REGION Network 6
   RUNG wire#powerrail
      #Module_Control(ReqUp := #Sequence_Control.ReqModulesUp, ReqDown := #Sequence_Control.ReqModulesDown, Sensor1Down := #Modules_DownPos1, Sensor1Up := #Modules_UpPos1, Sensor2Down := #Modules_DownPos2, Sensor2Up := #Modules_UpPos2, Interlock := true, Timeout :=, Valve => #Modules_Up, Error =>, "Step" =>, PosUp => #Module_Control.PosUp, PosDown => #Module_Control.PosDown)
   END_RUNG
   // the same network as SCL:
   #Module_Control(ReqUp := #Sequence_Control.ReqModulesUp,   // "CC_Vib_Modules"
                   ReqDown := #Sequence_Control.ReqModulesDown,
                   Sensor1Down := #Modules_DownPos1,
                   Sensor1Up := #Modules_UpPos1,
                   Sensor2Down := #Modules_DownPos2,
                   Sensor2Up := #Modules_UpPos2,
                   Interlock := true,
                   Valve => #Modules_Up,
                   PosUp => #Module_Control.PosUp,
                   PosDown => #Module_Control.PosDown);
END_REGION
END_FUNCTION_BLOCK

FUNCTION_BLOCK "CC_Sequence_Control"
{ S7_Optimized_Access := 'TRUE' }
VERSION : 0.1
   VAR_INPUT 
      Button_DriveRollers_Down : Bool;
      Button_DriveRollers_Up : Bool;
      Button_modules_Down : Bool;
      Button_modules_Up : Bool;
      Button_Pallete_Down : Bool;
      Button_Pallete_Up : Bool;
      Button_Wib : Bool;
      Seq_Forward : Bool;
      Seq_Backward : Bool;
      Drive_Rollers_DownPos : Bool;
      Drive_Rollers_UpPos : Bool;
      Pallete_DownPos : Bool;
      Pallete_UpPos : Bool;
      Modules_DownPos : Bool;
      Modules_UpPos : Bool;
      Centering_DownPos : Bool;
      Centering_UpPos : Bool;
   END_VAR

   VAR_OUTPUT 
      ReqPalleteUp : Bool;
      ReqPalleteDown : Bool;
      ReqDriveRollerUp : Bool;
      ReqDriveRollerDown : Bool;
      ReqModulesUp : Bool;
      ReqModulesDown : Bool;
      ReqVibrationEnable : Bool;
      Station_basePos : Bool;
   END_VAR

   VAR 
      Step { S7_SetPoint := 'True'} : Int;
      Button_Backward_TON {InstructionName := 'TON_TIME'; LibVersion := '1.0'} : TON_TIME;
   END_VAR

   VAR CONSTANT 
      sNOT_AUTOMATIC : Int;
      sBASE_POSITION : Int := 1;
      sMOVING_DRIVE_ROLLER : Int := 2;
      sMOVING_PALLETE : Int := 3;
      sMOVING_COMPACTION_MODULE : Int := 4;
      sCOMPACTING : Int := 5;
   END_VAR


BEGIN
	// Reset outputów
	#ReqPalleteUp := FALSE;
	#ReqPalleteDown := FALSE;
	#ReqDriveRollerUp := FALSE;
	#ReqDriveRollerDown := FALSE;
	#ReqVibrationEnable := FALSE;
	#ReqModulesUp := FALSE;
	#ReqModulesDown := FALSE;
	#Station_basePos := FALSE;
	
	IF #Button_DriveRollers_Down OR #Button_DriveRollers_Up OR #Button_Pallete_Down OR #Button_Pallete_Up OR #Button_modules_Down OR #Button_modules_Up OR #Button_Wib THEN
	    #Step := #sNOT_AUTOMATIC;
	ELSIF #Pallete_UpPos AND NOT #Seq_Forward AND #Drive_Rollers_UpPos AND #Modules_DownPos AND #Centering_DownPos THEN
	    #Step := #sBASE_POSITION;
	    #Station_basePos := true;
	END_IF;
	
	
	CASE #Step OF
	    #sBASE_POSITION:
	        IF #Seq_Forward THEN
	            #Step := #sMOVING_DRIVE_ROLLER;
	        END_IF;
	    #sMOVING_DRIVE_ROLLER:
	        #ReqPalleteUp := TRUE;
	        IF #Seq_Forward THEN
	            #ReqDriveRollerDown := TRUE;
	            IF #Drive_Rollers_DownPos THEN
	                #Step := #sMOVING_PALLETE;
	            END_IF;
	        ELSIF #Seq_Backward THEN
	            #ReqDriveRollerUp := TRUE;
	            IF #Drive_Rollers_UpPos THEN
	                #Step := #sBASE_POSITION;
	            END_IF;
	        END_IF;
	        
	    #sMOVING_PALLETE:
	        IF #Seq_Forward THEN
	            #ReqPalleteDown := TRUE;
	            IF #Pallete_DownPos THEN
	                #Step := #sMOVING_COMPACTION_MODULE;
	            END_IF;
	        ELSIF #Seq_Backward THEN
	            #ReqPalleteUp := TRUE;
	            IF #Pallete_UpPos THEN
	                #Step := #sMOVING_DRIVE_ROLLER;
	            END_IF;
	        END_IF;
	        
	    #sMOVING_COMPACTION_MODULE:
	        IF #Seq_Forward THEN
	            #ReqModulesUp := TRUE;
	         //   IF #Modules_UpPos THEN
	                #Step := #sCOMPACTING;
	         //   END_IF;
	        ELSIF #Seq_Backward THEN
	            #ReqModulesDown := TRUE;
	            IF #Modules_DownPos THEN
	                #Step := #sMOVING_PALLETE;
	            END_IF;
	        END_IF;
	        
	    #sCOMPACTING:
	        // Warunek zakończenia kompaktowania (np. czas lub czujnik)
	        IF #Seq_Forward THEN
	            #ReqVibrationEnable := TRUE;
	            #Step := #sCOMPACTING;
	        ELSIF #Seq_Backward THEN
	            #Step := #sMOVING_COMPACTION_MODULE;
	        END_IF;
	        
	    #sNOT_AUTOMATIC:
	        #ReqDriveRollerDown := #Button_DriveRollers_Down;
	        #ReqDriveRollerUp := #Button_DriveRollers_Up;
	        #ReqModulesDown := #Button_modules_Down;
	        #ReqModulesUp := #Button_modules_Up;
	        #ReqPalleteDown := #Button_Pallete_Down;
	        #ReqPalleteUp := #Button_Pallete_Up;
	        #ReqVibrationEnable := #Button_Wib;
	        
	END_CASE;
END_FUNCTION_BLOCK

FUNCTION_BLOCK "CC_Hydraulic_Rollers"   // FB101, LAD
{ S7_Optimized_Access := 'TRUE' }
// stored: AutoNumber false, MemoryReserve 100, SetENOAutomatically false
   VAR_INPUT
      ReqUp : Bool;
      ReqDown : Bool;
      Sensor1Down : Bool;
      Sensor1Up : Bool;
      Sensor2Down : Bool;
      Sensor2Up : Bool;
      InterlockMove : Bool;
      HydUnitReady : Bool;
   END_VAR
   VAR_OUTPUT
      HydraulicUnit : Bool;
      ValveUp : Bool;
      ValveDown : Bool;
      error : Byte;   // %X0 – nieprawidłowa pozycja dolna %X1 nieprawidłowa pozycja górna %X2 – przekroczony czas ruchu
      "Step" : Int;
      PosUp : Bool;
      PosDown : Bool;
   END_VAR
   VAR
      IEC_Extention { S7_SetPoint := 'True'} : TON_TIME;
      IEC_RETRACTION { S7_SetPoint := 'True'} : TON_TIME;
      tMotionTimeout { S7_SetPoint := 'True'} : TON_TIME;
   END_VAR
   VAR CONSTANT
      STEP_RETRACT : Int := 1;
      STEP_MOVING : Int := 2;
      STEP_EXTEND : Int := 3;
   END_VAR
BEGIN

REGION Network 1: ValveUp
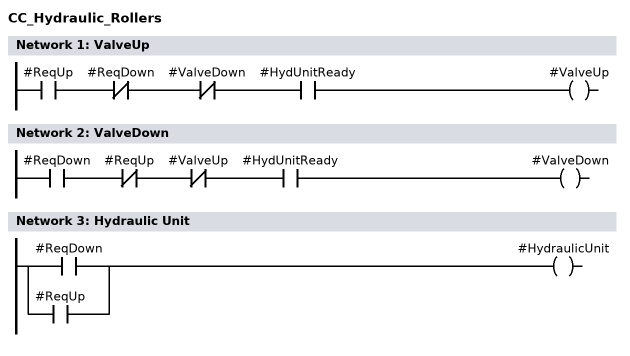
   RUNG wire#powerrail
      Contact( #ReqUp )
      I_Contact( #ReqDown )
      I_Contact( #ValveDown )
      Contact( #HydUnitReady )
      Coil( #ValveUp )
   END_RUNG
   // the same network as SCL:
   #ValveUp := #ReqUp AND NOT #ReqDown AND NOT #ValveDown AND #HydUnitReady;
END_REGION

REGION Network 2: ValveDown
   RUNG wire#powerrail
      Contact( #ReqDown )
      I_Contact( #ReqUp )
      I_Contact( #ValveUp )
      Contact( #HydUnitReady )
      Coil( #ValveDown )
   END_RUNG
   // the same network as SCL:
   #ValveDown := #ReqDown AND NOT #ReqUp AND NOT #ValveUp AND #HydUnitReady;
END_REGION

REGION Network 3: Hydraulic Unit
   RUNG wire#powerrail
      Contact( #ReqDown )
      wire#w1
      Coil( #HydraulicUnit )
   END_RUNG
   RUNG wire#powerrail
      Contact( #ReqUp )
   END_RUNG wire#w1
   // the same network as SCL:
   #HydraulicUnit := #ReqDown OR #ReqUp;
END_REGION

REGION Network 4 (SCL)
   #PosDown := false;
   #PosUp := FALSE;
   #Step := 0;
   IF #Sensor1Down = 0 AND #Sensor1Up = 1 AND #Sensor2Down = 0 AND #Sensor2Up = 1 THEN
       #Step.%X3 := TRUE;
       #PosUp := True;
   ELSIF #Sensor1Down = 1 AND #Sensor1Up =0 AND #Sensor2Down =1 AND #Sensor2Up =0 THEN
       #Step.%X1:= TRUE;
       #PosDown := True;
   ELSE
       #Step.%X2 := TRUE;
   END_IF;
END_REGION
END_FUNCTION_BLOCK

FUNCTION_BLOCK "CC_Pneumatic_Roller"   // FB104, LAD
{ S7_Optimized_Access := 'TRUE' }
// stored: AutoNumber false, MemoryReserve 100, SetENOAutomatically false
   VAR_INPUT
      ReqUp : Bool;
      ReqDown : Bool;
      Sensor1Down : Bool;
      Sensor1Up : Bool;
      Sensor2Down : Bool;
      Sensor2Up : Bool;
      Interlock : Bool;
      Timeout : Time := T#3s;
   END_VAR
   VAR_OUTPUT
      Valve : Bool;
      Error : Bool;
      "Step" : Int;
      PosUp : Bool;
      PosDown : Bool;
   END_VAR
   VAR
      IEC_Timout_retracting { S7_SetPoint := 'True'} : TOF_TIME;
      IEC_Timout_extracting { S7_SetPoint := 'True'} : TON_TIME;
   END_VAR
   VAR CONSTANT
      STEP_RETRACT : Int := 1;
      STEP_MOVING : Int := 2;
      STEP_EXTEND : Int := 3;
   END_VAR
BEGIN

REGION Network 1
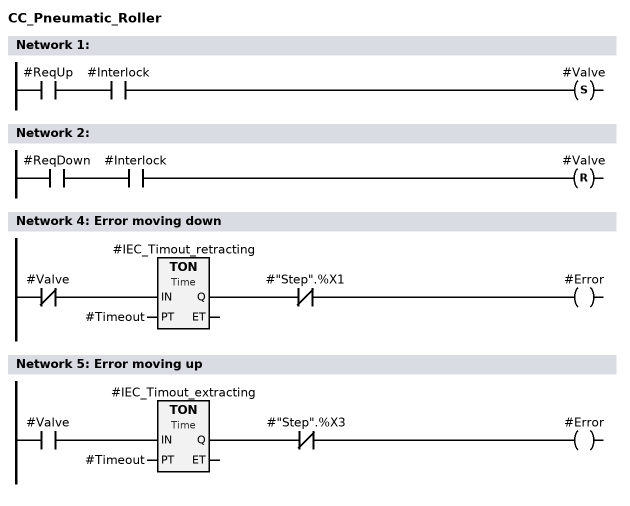
   RUNG wire#powerrail
      Contact( #ReqUp )
      Contact( #Interlock )
      S_Coil( #Valve )
   END_RUNG
   // the same network as SCL:
   IF #ReqUp AND #Interlock THEN #Valve := TRUE; END_IF;
END_REGION

REGION Network 2
   RUNG wire#powerrail
      Contact( #ReqDown )
      Contact( #Interlock )
      R_Coil( #Valve )
   END_RUNG
   // the same network as SCL:
   IF #ReqDown AND #Interlock THEN #Valve := FALSE; END_IF;
END_REGION

REGION Network 3 (SCL)
   #PosDown := FALSE;
   #PosUp := FALSE;
   #Step := 0;
   IF #Sensor1Down = 0 AND #Sensor1Up = 1 AND #Sensor2Down = 0 AND #Sensor2Up = 1 THEN
       #Step.%X3 :=1;
       #PosUp := True;
   ELSIF #Sensor1Down AND #Sensor1Up = 0 AND #Sensor2Down AND #Sensor2Up = 0 THEN
       #Step.%X1 := 1;
       #PosDown := True;
   ELSE
       #Step.%X2:= 1;
   END_IF;
END_REGION

REGION Network 4: Error moving down
   RUNG wire#powerrail
      I_Contact( #Valve )
      { S7_Templates := "time_type := Time" } #IEC_Timout_retracting.TON(pt := #Timeout, et =>)
      I_Contact( #"Step".%X1 )
      Coil( #Error )
   END_RUNG
   // the same network as SCL:
   #IEC_Timout_retracting(IN := NOT #Valve, PT := #Timeout);   // TON
   #Error := #IEC_Timout_retracting.Q AND NOT #"Step".%X1;
END_REGION

REGION Network 5: Error moving up
   RUNG wire#powerrail
      Contact( #Valve )
      { S7_Templates := "time_type := Time" } #IEC_Timout_extracting.TON(pt := #Timeout, et =>)
      I_Contact( #"Step".%X3 )
      Coil( #Error )
   END_RUNG
   // the same network as SCL:
   #IEC_Timout_extracting(IN := #Valve, PT := #Timeout);   // TON
   #Error := #IEC_Timout_extracting.Q AND NOT #"Step".%X3;
END_REGION
END_FUNCTION_BLOCK

FUNCTION_BLOCK "CC_Vib_Modules"   // FB102, LAD
{ S7_Optimized_Access := 'TRUE' }
// stored: AutoNumber false, MemoryReserve 100, SetENOAutomatically false
   VAR_INPUT
      ReqUp : Bool;
      ReqDown : Bool;
      Sensor1Down : Bool;
      Sensor1Up : Bool;
      Sensor2Down : Bool;
      Sensor2Up : Bool;
      Interlock : Bool := false;
      Timeout : Time := T#3s;
   END_VAR
   VAR_OUTPUT
      Valve : Bool;
      Error : Bool;
      "Step" : Int;
      PosUp : Bool;
      PosDown : Bool;
   END_VAR
   VAR
      IEC_Timout_retracting { S7_SetPoint := 'True'} : TOF_TIME;
      IEC_Timout_extracting { S7_SetPoint := 'True'} : TON_TIME;
   END_VAR
   VAR CONSTANT
      STEP_RETRACT : Int := 1;
      STEP_MOVING : Int := 2;
      STEP_EXTEND : Int := 3;
   END_VAR
BEGIN

REGION Network 1
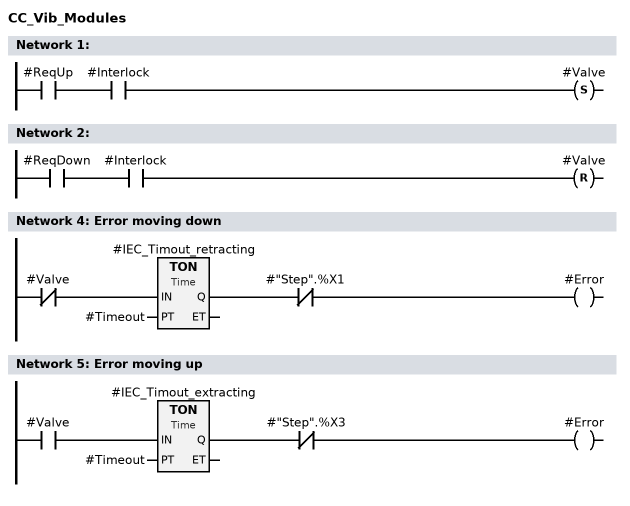
   RUNG wire#powerrail
      Contact( #ReqUp )
      Contact( #Interlock )
      S_Coil( #Valve )
   END_RUNG
   // the same network as SCL:
   IF #ReqUp AND #Interlock THEN #Valve := TRUE; END_IF;
END_REGION

REGION Network 2
   RUNG wire#powerrail
      Contact( #ReqDown )
      Contact( #Interlock )
      R_Coil( #Valve )
   END_RUNG
   // the same network as SCL:
   IF #ReqDown AND #Interlock THEN #Valve := FALSE; END_IF;
END_REGION

REGION Network 3 (SCL)
   #PosDown := false;
   #PosUp := false;
   #Step := 0;
   IF #Sensor1Down = 0 AND #Sensor1Up = 1 AND #Sensor2Down = 0 AND #Sensor2Up = 1 THEN
       #Step.%X3 := TRUE;
       #PosUp := True;
   ELSIF #Sensor1Down AND #Sensor1Up AND #Sensor2Down AND #Sensor2Up THEN
       #Step.%X1 := TRUE;
       #PosDown := True;
   ELSE
       #Step.%X2 := TRUE;
   END_IF;
END_REGION

REGION Network 4: Error moving down
   RUNG wire#powerrail
      I_Contact( #Valve )
      { S7_Templates := "time_type := Time" } #IEC_Timout_retracting.TON(pt := #Timeout, et =>)
      I_Contact( #"Step".%X1 )
      Coil( #Error )
   END_RUNG
   // the same network as SCL:
   #IEC_Timout_retracting(IN := NOT #Valve, PT := #Timeout);   // TON
   #Error := #IEC_Timout_retracting.Q AND NOT #"Step".%X1;
END_REGION

REGION Network 5: Error moving up
   RUNG wire#powerrail
      Contact( #Valve )
      { S7_Templates := "time_type := Time" } #IEC_Timout_extracting.TON(pt := #Timeout, et =>)
      I_Contact( #"Step".%X3 )
      Coil( #Error )
   END_RUNG
   // the same network as SCL:
   #IEC_Timout_extracting(IN := #Valve, PT := #Timeout);   // TON
   #Error := #IEC_Timout_extracting.Q AND NOT #"Step".%X3;
END_REGION
END_FUNCTION_BLOCK

FUNCTION_BLOCK "CC_Vibrator_Control"   // FB103, LAD
{ S7_Optimized_Access := 'TRUE' }
// stored: AutoNumber false, MemoryReserve 100, SetENOAutomatically false
   VAR_INPUT
      StartVibrating : Bool;
      Reset : Bool;
      Axis : TO_SpeedAxis;
      tmpVelocity : LReal := 2840.0;
   END_VAR
   VAR
      MC_Power_data { S7_SetPoint := 'True'} : MC_POWER;
      MC_Reset_data { S7_SetPoint := 'True'} : MC_RESET;
      MC_MoveJog_data { S7_SetPoint := 'True'} : MC_MOVEJOG;
      MC_HALT_data { S7_SetPoint := 'True'} : MC_HALT;
   END_VAR
BEGIN

REGION Network 1: Hydraulic Unit Motion Control
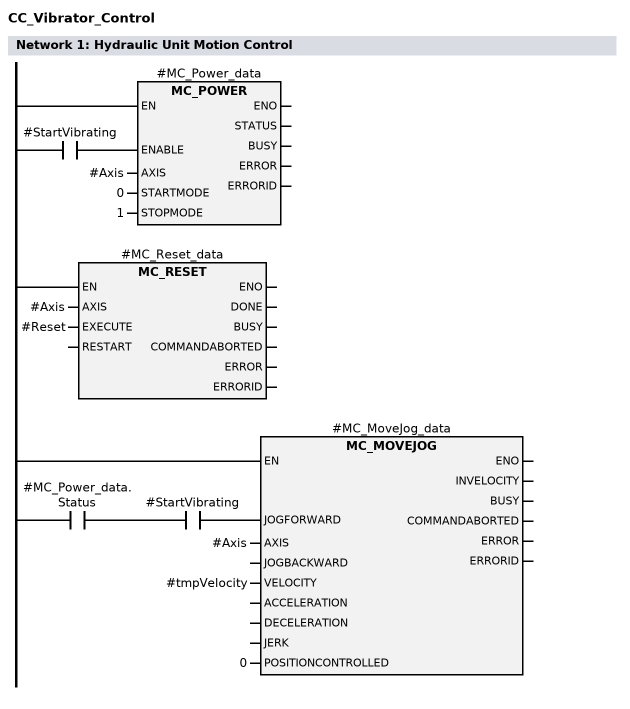
   RUNG wire#powerrail
      #MC_Power_data.MC_POWER(Enable := wire#w1, Axis := #Axis, StartMode := 0, StopMode := 1, Status =>, Busy =>, Error =>, ErrorId =>)
   END_RUNG
   RUNG wire#powerrail
      Contact( #StartVibrating )
   END_RUNG wire#w1
   RUNG wire#powerrail
      #MC_Reset_data.MC_RESET(Axis := #Axis, Execute := #Reset, Restart :=, Done =>, Busy =>, CommandAborted =>, Error =>, ErrorId =>)
   END_RUNG
   RUNG wire#powerrail
      #MC_MoveJog_data.MC_MOVEJOG(JogForward := wire#w2, Axis := #Axis, JogBackward :=, Velocity := #tmpVelocity, Acceleration :=, Deceleration :=, Jerk :=, PositionControlled := 0, InVelocity =>, Busy =>, CommandAborted =>, Error =>, ErrorId =>)
   END_RUNG
   RUNG wire#powerrail
      Contact( #MC_Power_data.Status )
      Contact( #StartVibrating )
   END_RUNG wire#w2
   // the same network as SCL:
   #MC_Power_data(Enable := #StartVibrating, Axis := #Axis, StartMode := 0, StopMode := 1);   // MC_POWER
   #MC_Reset_data(Axis := #Axis, Execute := #Reset);   // MC_RESET
   #MC_MoveJog_data(JogForward := #MC_Power_data.Status AND #StartVibrating,   // MC_MOVEJOG
                    Axis := #Axis,
                    Velocity := #tmpVelocity,
                    PositionControlled := 0);
END_REGION
END_FUNCTION_BLOCK

FUNCTION_BLOCK "Oil"   // FB8, LAD
{ S7_Optimized_Access := 'TRUE' }
// stored: MemoryReserve 100, SetENOAutomatically false
   VAR_INPUT
      Safety_OK : Bool;
      Pump_status : Bool;
      Pump_error : Bool;
      Pallette_Moving : Bool;
   END_VAR
   VAR_OUTPUT
      Pump : Bool;
      Main_Valve : Bool;
      Preparation_Valve : Bool;
      Nozzle_Valve : Bool;
      Pump_Volume_Output : Int;
   END_VAR
   VAR
      Pump_Reset { S7_SetPoint := 'True'} : TON_TIME;
      Pump_Volume { S7_SetPoint := 'True'} : Real;
      Oil_Station_Enable : Bool;
   END_VAR
   VAR_TEMP
      tmp : Int;
   END_VAR
BEGIN

REGION Network 1
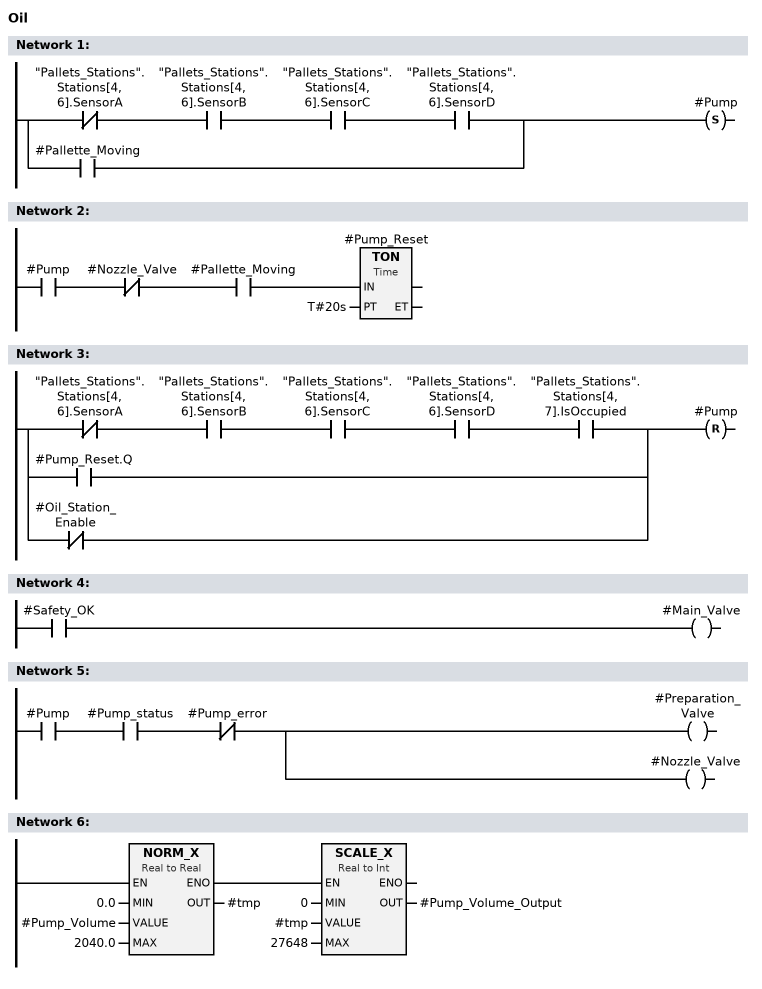
   RUNG wire#powerrail
      I_Contact( "Pallets_Stations".Stations[4, 6].SensorA )
      Contact( "Pallets_Stations".Stations[4, 6].SensorB )
      Contact( "Pallets_Stations".Stations[4, 6].SensorC )
      Contact( "Pallets_Stations".Stations[4, 6].SensorD )
      wire#w1
      S_Coil( #Pump )
   END_RUNG
   RUNG wire#powerrail
      Contact( #Pallette_Moving )
   END_RUNG wire#w1
   // the same network as SCL:
   IF (NOT "Pallets_Stations".Stations[4, 6].SensorA AND "Pallets_Stations".Stations[4, 6].SensorB AND "Pallets_Stations".Stations[4, 6].SensorC AND "Pallets_Stations".Stations[4, 6].SensorD) OR #Pallette_Moving THEN
       #Pump := TRUE;
   END_IF;
END_REGION

REGION Network 2
   RUNG wire#powerrail
      Contact( #Pump )
      I_Contact( #Nozzle_Valve )
      Contact( #Pallette_Moving )
      { S7_Templates := "time_type := Time" } #Pump_Reset.TON(pt := T#20s, et =>)
   END_RUNG
   // the same network as SCL:
   #Pump_Reset(IN := #Pump AND NOT #Nozzle_Valve AND #Pallette_Moving, PT := T#20s);   // TON
END_REGION

REGION Network 3
   RUNG wire#powerrail
      I_Contact( "Pallets_Stations".Stations[4, 6].SensorA )
      Contact( "Pallets_Stations".Stations[4, 6].SensorB )
      Contact( "Pallets_Stations".Stations[4, 6].SensorC )
      Contact( "Pallets_Stations".Stations[4, 6].SensorD )
      Contact( "Pallets_Stations".Stations[4, 7].IsOccupied )
      wire#w1
      R_Coil( #Pump )
   END_RUNG
   RUNG wire#powerrail
      Contact( #Pump_Reset.Q )
   END_RUNG wire#w1
   RUNG wire#powerrail
      I_Contact( #Oil_Station_Enable )
   END_RUNG wire#w1
   // the same network as SCL:
   IF (NOT "Pallets_Stations".Stations[4, 6].SensorA AND "Pallets_Stations".Stations[4, 6].SensorB AND "Pallets_Stations".Stations[4, 6].SensorC AND "Pallets_Stations".Stations[4, 6].SensorD AND "Pallets_Stations".Stations[4, 7].IsOccupied) OR #Pump_Reset.Q OR NOT #Oil_Station_Enable THEN
       #Pump := FALSE;
   END_IF;
END_REGION

REGION Network 4
   RUNG wire#powerrail
      Contact( #Safety_OK )
      Coil( #Main_Valve )
   END_RUNG
   // the same network as SCL:
   #Main_Valve := #Safety_OK;
END_REGION

REGION Network 5
   RUNG wire#powerrail
      Contact( #Pump )
      Contact( #Pump_status )
      I_Contact( #Pump_error )
      wire#w1
      Coil( #Preparation_Valve )
   END_RUNG
   RUNG wire#w1
      Coil( #Nozzle_Valve )
   END_RUNG
   // the same network as SCL:
   #Preparation_Valve := #Pump AND #Pump_status AND NOT #Pump_error;
   #Nozzle_Valve := #Preparation_Valve;
END_REGION

REGION Network 6
   RUNG wire#powerrail
      { S7_Templates := "[SrcType := Real, DestType := Real]" } Normalize(min := 0.0, value := #Pump_Volume, max := 2040.0, out => #tmp)
      { S7_Templates := "[SrcType := Real, DestType := Int]" } Scale(min := 0, value := #tmp, max := 27648, out => #Pump_Volume_Output)
   END_RUNG
   // the same network as SCL:
   #tmp := NORM_X(MIN := 0.0, VALUE := #Pump_Volume, MAX := 2040.0);
   #Pump_Volume_Output := SCALE_X(MIN := 0, VALUE := #tmp, MAX := 27648);
END_REGION
END_FUNCTION_BLOCK

FUNCTION_BLOCK "HMI_Test"
{ S7_Optimized_Access := 'TRUE' }
VERSION : 0.1
   VAR 
      Old_Value : USInt;
      HMI_Connection_Alarm : Bool;
      Timer_2s {InstructionName := 'TON_TIME'; LibVersion := '1.0'; S7_SetPoint := 'False'} : TON_TIME;
   END_VAR


BEGIN
	IF #Timer_2s.Q THEN
	    #HMI_Connection_Alarm := ("HMI_DB".Heart_Bit = #Old_Value);
	    #Old_Value := "HMI_DB".Heart_Bit;
	END_IF;
	
	#Timer_2s(IN := NOT #Timer_2s.Q,
	          PT := T#2s);
	
END_FUNCTION_BLOCK

ORGANIZATION_BLOCK "CyclicInterrupt"   // OB30, LAD, CyclicInterrupt
{ S7_Optimized_Access := 'TRUE' }
// stored: SetENOAutomatically false
   VAR_INPUT
      Initial_Call : Bool;   // Initial call of this OB
      Event_Count : Int;   // Events discarded
   END_VAR
BEGIN

REGION Network 1
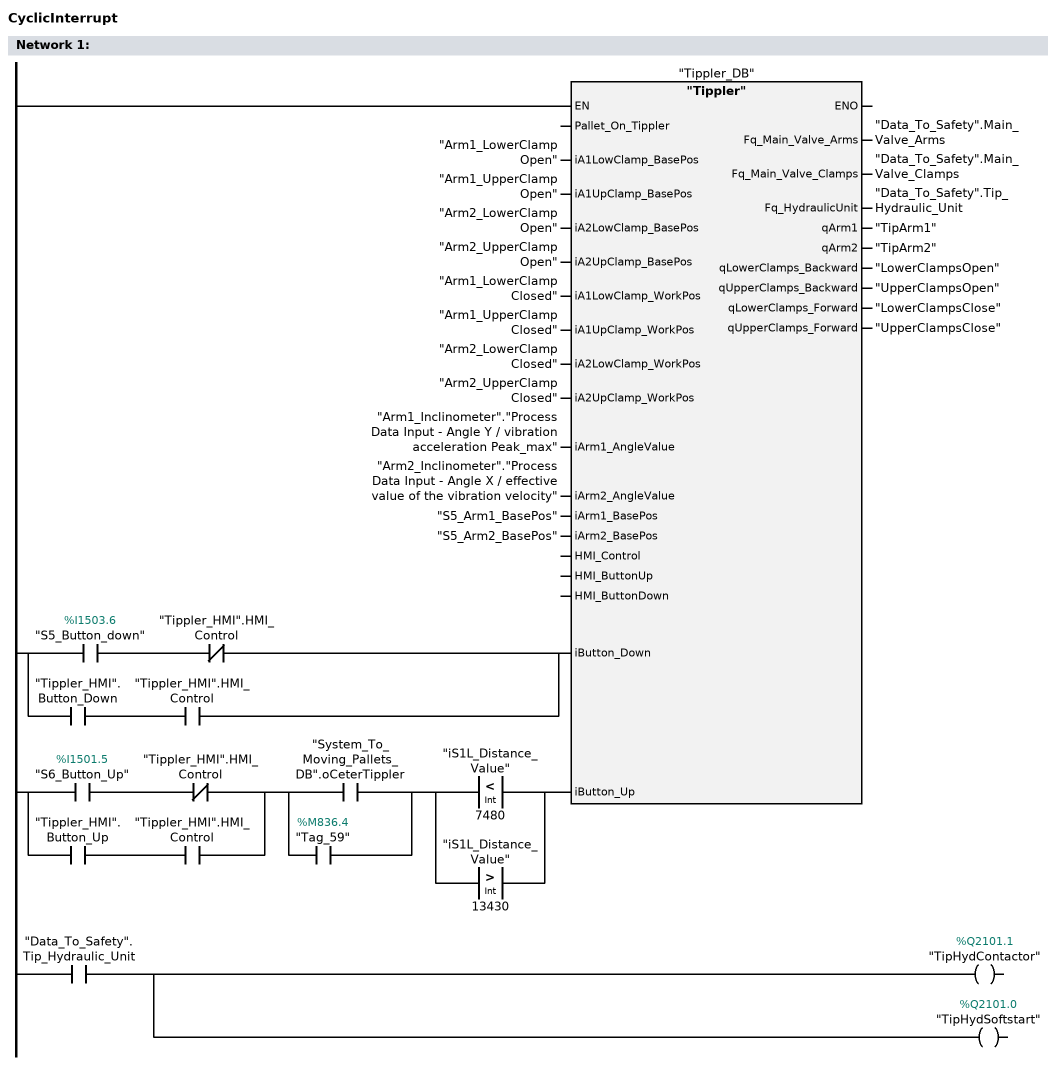
   RUNG wire#powerrail
      "Tippler_DB"(iButton_Down := wire#w1, iButton_Up := wire#w4, Pallet_On_Tippler :=, iA1LowClamp_BasePos := "Arm1_LowerClampOpen", iA1UpClamp_BasePos := "Arm1_UpperClampOpen", iA2LowClamp_BasePos := "Arm2_LowerClampOpen", iA2UpClamp_BasePos := "Arm2_UpperClampOpen", iA1LowClamp_WorkPos := "Arm1_LowerClampClosed", iA1UpClamp_WorkPos := "Arm1_UpperClampClosed", iA2LowClamp_WorkPos := "Arm2_LowerClampClosed", iA2UpClamp_WorkPos := "Arm2_UpperClampClosed", iArm1_AngleValue := "Arm1_Inclinometer"."Process Data Input - Angle Y / vibration acceleration Peak_max", iArm2_AngleValue := "Arm2_Inclinometer"."Process Data Input - Angle X / effective value of the vibration velocity", iArm1_BasePos := "S5_Arm1_BasePos", iArm2_BasePos := "S5_Arm2_BasePos", HMI_Control :=, HMI_ButtonUp :=, HMI_ButtonDown :=, Fq_Main_Valve_Arms => "Data_To_Safety".Main_Valve_Arms, Fq_Main_Valve_Clamps => "Data_To_Safety".Main_Valve_Clamps, Fq_HydraulicUnit => "Data_To_Safety".Tip_Hydraulic_Unit, qArm1 => "TipArm1", qArm2 => "TipArm2", qLowerClamps_Backward => "LowerClampsOpen", qUpperClamps_Backward => "UpperClampsOpen", qLowerClamps_Forward => "LowerClampsClose", qUpperClamps_Forward => "UpperClampsClose")
   END_RUNG
   RUNG wire#powerrail
      Contact( "S5_Button_down" )
      I_Contact( "Tippler_HMI".HMI_Control )
   END_RUNG wire#w1
   RUNG wire#powerrail
      Contact( "Tippler_HMI".Button_Down )
      Contact( "Tippler_HMI".HMI_Control )
   END_RUNG wire#w1
   RUNG wire#powerrail
      Contact( "S6_Button_Up" )
      I_Contact( "Tippler_HMI".HMI_Control )
      wire#w2
      Contact( "System_To_Moving_Pallets_DB".oCeterTippler )
      wire#w3
      { S7_Templates := "SrcType := Int" } LT_Contact(in1 := "iS1L_Distance_Value", in2 := 7480)
   END_RUNG wire#w4
   RUNG wire#powerrail
      Contact( "Tippler_HMI".Button_Up )
      Contact( "Tippler_HMI".HMI_Control )
   END_RUNG wire#w2
   RUNG wire#w2
      Contact( "Tag_59" )
   END_RUNG wire#w3
   RUNG wire#w3
      { S7_Templates := "SrcType := Int" } GT_Contact(in1 := "iS1L_Distance_Value", in2 := 13430)
   END_RUNG wire#w4
   RUNG wire#powerrail
      Contact( "Data_To_Safety".Tip_Hydraulic_Unit )
      wire#w5
      Coil( "TipHydContactor" )
   END_RUNG
   RUNG wire#w5
      Coil( "TipHydSoftstart" )
   END_RUNG
   // the same network as SCL:
   "Tippler_DB"(iA1LowClamp_BasePos := "Arm1_LowerClampOpen",   // "Tippler"
                iA1UpClamp_BasePos := "Arm1_UpperClampOpen",
                iA2LowClamp_BasePos := "Arm2_LowerClampOpen",
                iA2UpClamp_BasePos := "Arm2_UpperClampOpen",
                iA1LowClamp_WorkPos := "Arm1_LowerClampClosed",
                iA1UpClamp_WorkPos := "Arm1_UpperClampClosed",
                iA2LowClamp_WorkPos := "Arm2_LowerClampClosed",
                iA2UpClamp_WorkPos := "Arm2_UpperClampClosed",
                iArm1_AngleValue := "Arm1_Inclinometer"."Process Data Input - Angle Y / vibration acceleration Peak_max",
                iArm2_AngleValue := "Arm2_Inclinometer"."Process Data Input - Angle X / effective value of the vibration velocity",
                iArm1_BasePos := "S5_Arm1_BasePos",
                iArm2_BasePos := "S5_Arm2_BasePos",
                iButton_Down := ("S5_Button_down" AND NOT "Tippler_HMI".HMI_Control) OR ("Tippler_HMI".Button_Down AND "Tippler_HMI".HMI_Control),
                iButton_Up := (("S6_Button_Up" AND NOT "Tippler_HMI".HMI_Control) OR ("Tippler_HMI".Button_Up AND "Tippler_HMI".HMI_Control)) AND ("System_To_Moving_Pallets_DB".oCeterTippler OR "Tag_59") AND (("iS1L_Distance_Value" < 7480) OR ("iS1L_Distance_Value" > 13430)),
                Fq_Main_Valve_Arms => "Data_To_Safety".Main_Valve_Arms,
                Fq_Main_Valve_Clamps => "Data_To_Safety".Main_Valve_Clamps,
                Fq_HydraulicUnit => "Data_To_Safety".Tip_Hydraulic_Unit,
                qArm1 => "TipArm1",
                qArm2 => "TipArm2",
                qLowerClamps_Backward => "LowerClampsOpen",
                qUpperClamps_Backward => "UpperClampsOpen",
                qLowerClamps_Forward => "LowerClampsClose",
                qUpperClamps_Forward => "UpperClampsClose");
   "TipHydContactor" := "Data_To_Safety".Tip_Hydraulic_Unit;
   "TipHydSoftstart" := "Data_To_Safety".Tip_Hydraulic_Unit;
END_REGION
END_ORGANIZATION_BLOCK

FUNCTION_BLOCK "Tippler"   // FB400, LAD
{ S7_Optimized_Access := 'TRUE' }
// stored: AutoNumber false, MemoryReserve 100, SetENOAutomatically false
   VAR_INPUT
      Pallet_On_Tippler : Bool;
      iA1LowClamp_BasePos : Bool;
      iA1UpClamp_BasePos : Bool;
      iA2LowClamp_BasePos : Bool;
      iA2UpClamp_BasePos : Bool;
      iA1LowClamp_WorkPos : Bool;
      iA1UpClamp_WorkPos : Bool;
      iA2LowClamp_WorkPos : Bool;
      iA2UpClamp_WorkPos : Bool;
      iArm1_AngleValue : Int;
      iArm2_AngleValue : Int;
      iArm1_BasePos : Bool;
      iArm2_BasePos : Bool;
      HMI_Control : Bool;
      HMI_ButtonUp : Bool;
      HMI_ButtonDown : Bool;
      iButton_Down : Bool;
      iButton_Up : Bool;
   END_VAR
   VAR_OUTPUT
      Fq_Main_Valve_Arms : Bool;
      Fq_Main_Valve_Clamps : Bool;
      Fq_HydraulicUnit : Bool;
      qArm1 : Int;
      qArm2 : Int;
      qLowerClamps_Backward : Bool;
      qUpperClamps_Backward : Bool;
      qLowerClamps_Forward : Bool;
      qUpperClamps_Forward : Bool;
   END_VAR
   VAR
      Hydraulic_Ready { S7_SetPoint := 'True'} : TON_TIME;
      Hydraulic_Off { S7_SetPoint := 'True'} : TON_TIME;
      LowerClamps { S7_SetPoint := 'True'} : "Clamp";
      UpperClamps { S7_SetPoint := 'True'} : "Clamp";
      Arms { S7_SetPoint := 'True'} : "Arms";
      "Step" { S7_SetPoint := 'True'} : Int;
      ReqArmsDown : Bool;
      ReqArmsUp : Bool;
      Arms_workPos : Bool;
      Arms_basePos : Bool;
      Arms_clampsOperPos { S7_SetPoint := 'True'} : Bool;
      Tippler_maintenance { S7_SetPoint := 'True'} : "Tippler_maintenance";
      ButtonArmsDown { S7_SetPoint := 'True'} : Bool;
      ButtonArmsUp { S7_SetPoint := 'True'} : Bool;
      ReqLowerClampsClose : Bool;
      ReqUpperClampsClose : Bool;
      ReqLowerClampsOpen : Bool;
      ReqUpperClampsOpen : Bool;
      Timer_ClampsWorkPos { S7_SetPoint := 'True'} : TON_TIME;
      Timer_ClampsBasePos { S7_SetPoint := 'True'} : TON_TIME;
      Tippler_keep_down { S7_SetPoint := 'True'} : TP_TIME;
      N_Trig_Button_Down { S7_SetPoint := 'True'} : Bool;
   END_VAR
   VAR_TEMP
      Arm_Valves_Not_Actuated : Bool;
      Clamp_Valves_Not_Actuated : Bool;
   END_VAR
   VAR_TEMP   // added for the SCL form of the ladder/FBD networks
      _w1 : Bool;
   END_VAR
BEGIN

REGION Network 1: Zawory na ramionach niewysterowane
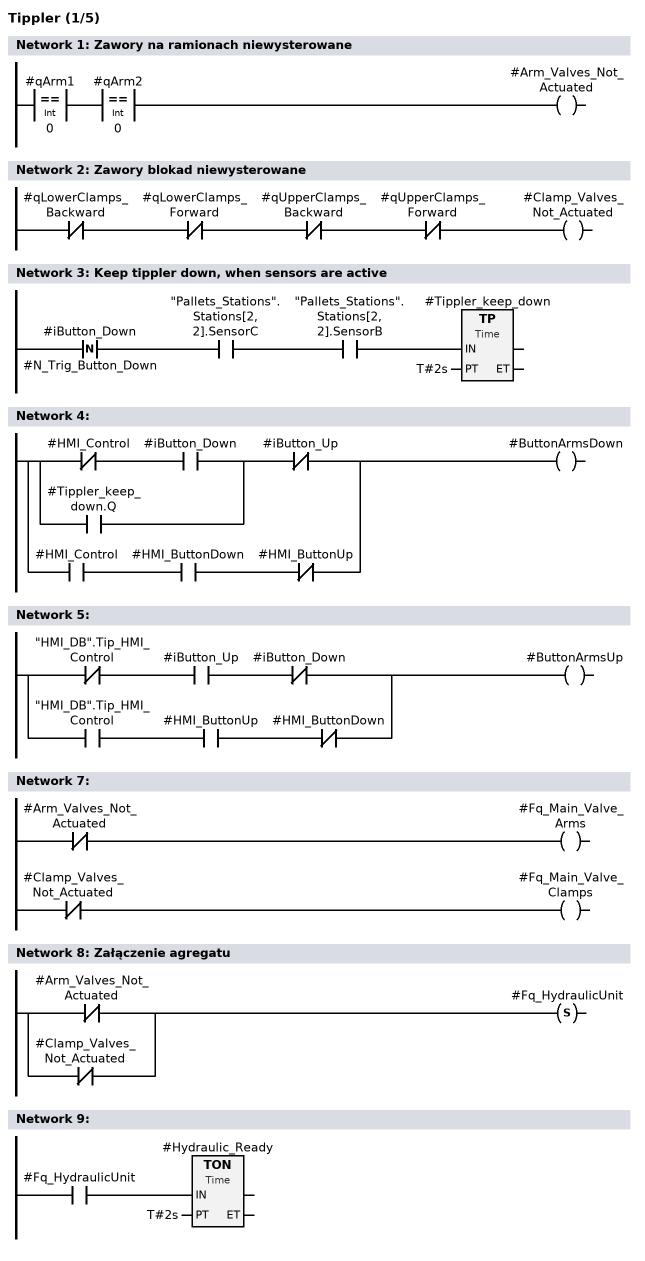
   RUNG wire#powerrail
      { S7_Templates := "SrcType := Int" } EQ_Contact(in1 := #qArm1, in2 := 0)
      { S7_Templates := "SrcType := Int" } EQ_Contact(in1 := #qArm2, in2 := 0)
      Coil( #Arm_Valves_Not_Actuated )
   END_RUNG
   // the same network as SCL:
   #Arm_Valves_Not_Actuated := (#qArm1 = 0) AND (#qArm2 = 0);
END_REGION

REGION Network 2: Zawory blokad niewysterowane
   RUNG wire#powerrail
      I_Contact( #qLowerClamps_Backward )
      I_Contact( #qLowerClamps_Forward )
      I_Contact( #qUpperClamps_Backward )
      I_Contact( #qUpperClamps_Forward )
      Coil( #Clamp_Valves_Not_Actuated )
   END_RUNG
   // the same network as SCL:
   #Clamp_Valves_Not_Actuated := NOT #qLowerClamps_Backward AND NOT #qLowerClamps_Forward AND NOT #qUpperClamps_Backward AND NOT #qUpperClamps_Forward;
END_REGION

REGION Network 3: Keep tippler down, when sensors are active
   RUNG wire#powerrail
      N_Contact(operand := #iButton_Down, bit := #N_Trig_Button_Down)
      Contact( "Pallets_Stations".Stations[2, 2].SensorC )
      Contact( "Pallets_Stations".Stations[2, 2].SensorB )
      { S7_Templates := "time_type := Time" } #Tippler_keep_down.TP(pt := T#2s, et =>)
   END_RUNG
   // the same network as SCL:
   #_w1 := NOT #iButton_Down AND #N_Trig_Button_Down;   // falling edge of #iButton_Down
   #N_Trig_Button_Down := #iButton_Down;
   #Tippler_keep_down(IN := #_w1 AND "Pallets_Stations".Stations[2, 2].SensorC AND "Pallets_Stations".Stations[2, 2].SensorB,   // TP
                      PT := T#2s);
END_REGION

REGION Network 4
   RUNG wire#powerrail
      I_Contact( #HMI_Control )
      Contact( #iButton_Down )
      wire#w1
      I_Contact( #iButton_Up )
      wire#w2
      Coil( #ButtonArmsDown )
   END_RUNG
   RUNG wire#powerrail
      Contact( #Tippler_keep_down.Q )
   END_RUNG wire#w1
   RUNG wire#powerrail
      Contact( #HMI_Control )
      Contact( #HMI_ButtonDown )
      I_Contact( #HMI_ButtonUp )
   END_RUNG wire#w2
   // the same network as SCL:
   #ButtonArmsDown := (((NOT #HMI_Control AND #iButton_Down) OR #Tippler_keep_down.Q) AND NOT #iButton_Up) OR (#HMI_Control AND #HMI_ButtonDown AND NOT #HMI_ButtonUp);
END_REGION

REGION Network 5
   RUNG wire#powerrail
      I_Contact( "HMI_DB".Tip_HMI_Control )
      Contact( #iButton_Up )
      I_Contact( #iButton_Down )
      wire#w1
      Coil( #ButtonArmsUp )
   END_RUNG
   RUNG wire#powerrail
      Contact( "HMI_DB".Tip_HMI_Control )
      Contact( #HMI_ButtonUp )
      I_Contact( #HMI_ButtonDown )
   END_RUNG wire#w1
   // the same network as SCL:
   #ButtonArmsUp := (NOT "HMI_DB".Tip_HMI_Control AND #iButton_Up AND NOT #iButton_Down) OR ("HMI_DB".Tip_HMI_Control AND #HMI_ButtonUp AND NOT #HMI_ButtonDown);
END_REGION

REGION Network 6 (SCL)
   #ReqArmsDown := 0;
   #ReqArmsUp := 0;
   #ReqLowerClampsClose := 0;
   #ReqUpperClampsClose := 0;
   #ReqLowerClampsOpen := 0;
   #ReqUpperClampsOpen := 0;
   IF "HMI_DB".Tip_MT_Control = 1 THEN
       #Step := 0;
   END_IF;
   CASE #Step OF
       0:
           IF #ButtonArmsDown THEN
               IF #Arms_basePos = 0 AND #iA1LowClamp_BasePos AND #iA2LowClamp_BasePos AND #iA1UpClamp_BasePos AND #iA2UpClamp_BasePos THEN
                   #ReqArmsDown := 1;
               ELSIF #Arms_basePos = 0 AND #Arms_clampsOperPos = 0 AND (#Arms.Arm1AngleValue > 3 OR  #Arms.Arm2AngleValue > 3) THEN
                   #ReqArmsDown := 1;
               ELSIF #Arms_clampsOperPos OR #Arms_basePos OR #Pallet_On_Tippler = 0 THEN
                   IF #iA1LowClamp_BasePos = 0 OR #iA2LowClamp_BasePos = 0 THEN
                       #ReqLowerClampsOpen := 1;
                   END_IF;
                   IF #iA1UpClamp_BasePos = 0 OR #iA2UpClamp_BasePos = 0 THEN
                       #ReqUpperClampsOpen := 1;
                   END_IF;
               END_IF;
               IF  #iA1LowClamp_BasePos AND #iA1UpClamp_BasePos AND #iA2LowClamp_BasePos AND #iA2UpClamp_BasePos THEN
                   #Step += 1;
               END_IF;
           END_IF;

           1:
               IF #ButtonArmsUp AND NOT #Arms_clampsOperPos AND #Arms.Arm1AngleValue < 4 AND #Arms.Arm2AngleValue < 4 THEN
                   #ReqArmsUp := 1;
               ELSIF #ButtonArmsDown AND #Arms_basePos = 0 THEN
                   #ReqArmsDown := 1;
               ELSIF #ButtonArmsUp AND #Arms_clampsOperPos THEN
                   //#ReqArmsUp := 0;
                   #Step += 1;
               END_IF;

       2:
           IF #ButtonArmsUp AND #Arms.Arm1AngleValue < 12 AND #Arms.Arm2AngleValue < 12 THEN
               IF NOT #Timer_ClampsWorkPos.Q THEN
                   #ReqUpperClampsClose := 1;
                   #ReqLowerClampsClose := 1;
                   #ReqArmsUp := 1;
               END_IF;
           ELSIF #ButtonArmsDown THEN
               IF #Timer_ClampsBasePos.Q = 0 THEN
                   #ReqLowerClampsOpen := 1;
                   #ReqUpperClampsOpen := 1;
               END_IF;
           END_IF;
           #Timer_ClampsWorkPos(IN:= #Step = 2 AND #ButtonArmsUp AND #iA1LowClamp_WorkPos AND #iA1UpClamp_WorkPos AND #iA2LowClamp_WorkPos AND #iA2UpClamp_WorkPos,
                                PT:=t#3s);
           IF (#Timer_ClampsWorkPos.Q) THEN
               #Step += 1;
           END_IF;
           #Timer_ClampsBasePos(IN:= #Step = 2 AND #ButtonArmsDown AND #iA1LowClamp_BasePos AND #iA1UpClamp_BasePos AND #iA2LowClamp_BasePos AND #iA2UpClamp_BasePos ,
                                PT:=t#3s);

           IF #Timer_ClampsBasePos.Q THEN
               #Step -= 1;
           END_IF;
       3:
           IF #ButtonArmsUp AND #Arms_workPos = 0 AND #iA1LowClamp_WorkPos AND #iA1UpClamp_WorkPos AND #iA2LowClamp_WorkPos AND #iA2UpClamp_WorkPos THEN
               #ReqArmsUp := 1;
           ELSIF #ButtonArmsDown AND #Arms_clampsOperPos = 0 AND #iA1LowClamp_WorkPos AND #iA1UpClamp_WorkPos AND #iA2LowClamp_WorkPos AND #iA2UpClamp_WorkPos THEN
               #ReqArmsDown := 1;
           ELSIF #ButtonArmsUp AND #Arms_workPos = 1 AND #iA1LowClamp_WorkPos AND #iA1UpClamp_WorkPos AND #iA2LowClamp_WorkPos AND #iA2UpClamp_WorkPos THEN
               #Step := 4;
           ELSIF #ButtonArmsDown AND #Arms_clampsOperPos THEN
               #ReqArmsDown := 0;
               #Step := 2;
           END_IF;
       4:
           IF #ButtonArmsDown AND #Arms_clampsOperPos = 0 AND #iA1LowClamp_WorkPos AND #iA1UpClamp_WorkPos AND #iA2LowClamp_WorkPos AND #iA2UpClamp_WorkPos THEN
               #Step := 3;
           END_IF;
       ELSE
           #Step := 0;
   END_CASE;
END_REGION

REGION Network 7
   RUNG wire#powerrail
      I_Contact( #Arm_Valves_Not_Actuated )
      Coil( #Fq_Main_Valve_Arms )
   END_RUNG
   RUNG wire#powerrail
      I_Contact( #Clamp_Valves_Not_Actuated )
      Coil( #Fq_Main_Valve_Clamps )
   END_RUNG
   // the same network as SCL:
   #Fq_Main_Valve_Arms := NOT #Arm_Valves_Not_Actuated;
   #Fq_Main_Valve_Clamps := NOT #Clamp_Valves_Not_Actuated;
END_REGION

REGION Network 8: Załączenie agregatu
   RUNG wire#powerrail
      I_Contact( #Arm_Valves_Not_Actuated )
      wire#w1
      S_Coil( #Fq_HydraulicUnit )
   END_RUNG
   RUNG wire#powerrail
      I_Contact( #Clamp_Valves_Not_Actuated )
   END_RUNG wire#w1
   // the same network as SCL:
   IF NOT #Arm_Valves_Not_Actuated OR NOT #Clamp_Valves_Not_Actuated THEN #Fq_HydraulicUnit := TRUE; END_IF;
END_REGION

REGION Network 9
   RUNG wire#powerrail
      Contact( #Fq_HydraulicUnit )
      { S7_Templates := "time_type := Time" } #Hydraulic_Ready.TON(pt := T#2s, et =>)
   END_RUNG
   // the same network as SCL:
   #Hydraulic_Ready(IN := #Fq_HydraulicUnit, PT := T#2s);   // TON
END_REGION

REGION Network 10: Czasowe wyłączenie po braku działania
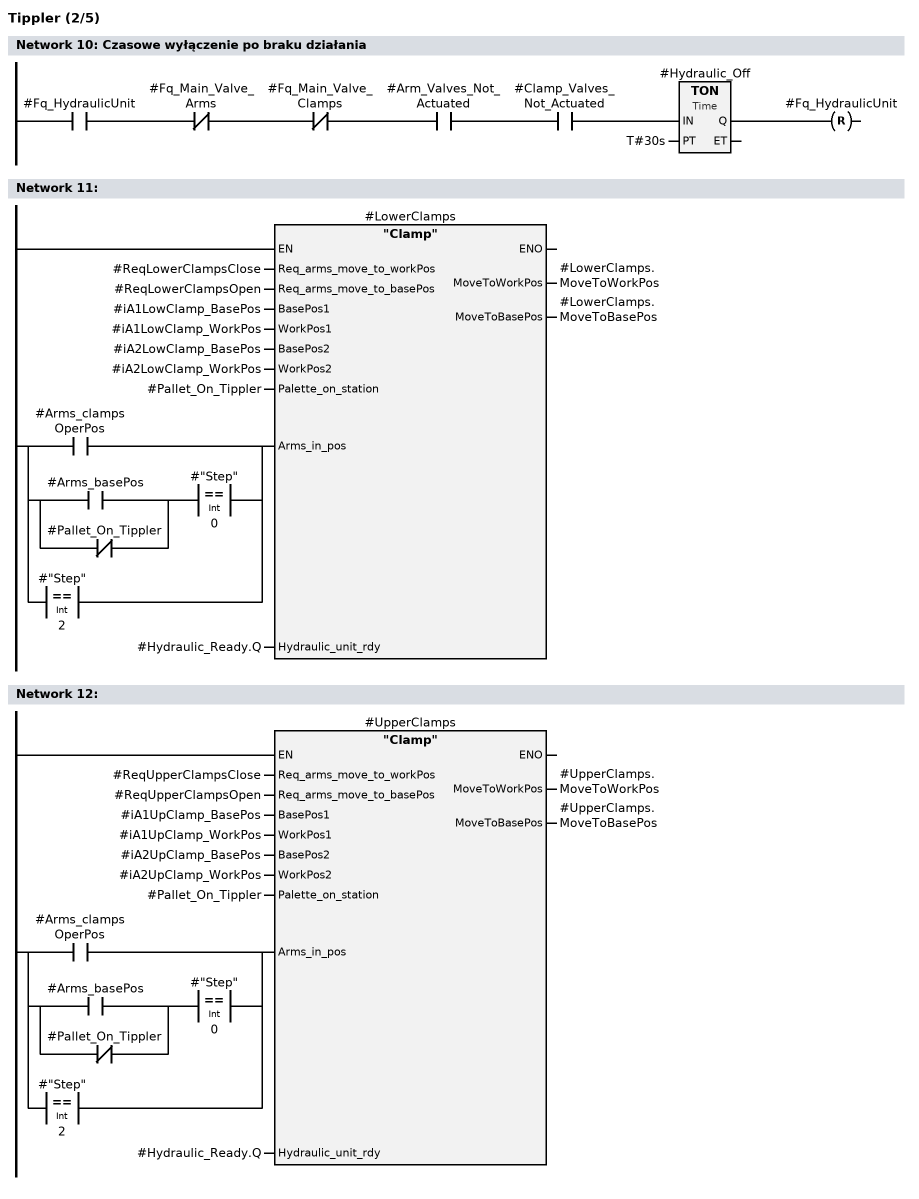
   RUNG wire#powerrail
      Contact( #Fq_HydraulicUnit )
      I_Contact( #Fq_Main_Valve_Arms )
      I_Contact( #Fq_Main_Valve_Clamps )
      Contact( #Arm_Valves_Not_Actuated )
      Contact( #Clamp_Valves_Not_Actuated )
      { S7_Templates := "time_type := Time" } #Hydraulic_Off.TON(pt := T#30s, et =>)
      R_Coil( #Fq_HydraulicUnit )
   END_RUNG
   // the same network as SCL:
   #Hydraulic_Off(IN := #Fq_HydraulicUnit AND NOT #Fq_Main_Valve_Arms AND NOT #Fq_Main_Valve_Clamps AND #Arm_Valves_Not_Actuated AND #Clamp_Valves_Not_Actuated,   // TON
                  PT := T#30s);
   IF #Hydraulic_Off.Q THEN #Fq_HydraulicUnit := FALSE; END_IF;
END_REGION

REGION Network 11
   RUNG wire#powerrail
      #LowerClamps(Arms_in_pos := wire#w2, Req_arms_move_to_workPos := #ReqLowerClampsClose, Req_arms_move_to_basePos := #ReqLowerClampsOpen, BasePos1 := #iA1LowClamp_BasePos, WorkPos1 := #iA1LowClamp_WorkPos, BasePos2 := #iA2LowClamp_BasePos, WorkPos2 := #iA2LowClamp_WorkPos, Palette_on_station := #Pallet_On_Tippler, Hydraulic_unit_rdy := #Hydraulic_Ready.Q, MoveToWorkPos => #LowerClamps.MoveToWorkPos, MoveToBasePos => #LowerClamps.MoveToBasePos)
   END_RUNG
   RUNG wire#powerrail
      Contact( #Arms_clampsOperPos )
   END_RUNG wire#w2
   RUNG wire#powerrail
      Contact( #Arms_basePos )
      wire#w1
      { S7_Templates := "SrcType := Int" } EQ_Contact(in1 := #"Step", in2 := 0)
   END_RUNG wire#w2
   RUNG wire#powerrail
      I_Contact( #Pallet_On_Tippler )
   END_RUNG wire#w1
   RUNG wire#powerrail
      { S7_Templates := "SrcType := Int" } EQ_Contact(in1 := #"Step", in2 := 2)
   END_RUNG wire#w2
   // the same network as SCL:
   #LowerClamps(Req_arms_move_to_workPos := #ReqLowerClampsClose,   // "Clamp"
                Req_arms_move_to_basePos := #ReqLowerClampsOpen,
                BasePos1 := #iA1LowClamp_BasePos,
                WorkPos1 := #iA1LowClamp_WorkPos,
                BasePos2 := #iA2LowClamp_BasePos,
                WorkPos2 := #iA2LowClamp_WorkPos,
                Palette_on_station := #Pallet_On_Tippler,
                Arms_in_pos := #Arms_clampsOperPos OR ((#Arms_basePos OR NOT #Pallet_On_Tippler) AND (#"Step" = 0)) OR (#"Step" = 2),
                Hydraulic_unit_rdy := #Hydraulic_Ready.Q,
                MoveToWorkPos => #LowerClamps.MoveToWorkPos,
                MoveToBasePos => #LowerClamps.MoveToBasePos);
END_REGION

REGION Network 12
   RUNG wire#powerrail
      #UpperClamps(Arms_in_pos := wire#w2, Req_arms_move_to_workPos := #ReqUpperClampsClose, Req_arms_move_to_basePos := #ReqUpperClampsOpen, BasePos1 := #iA1UpClamp_BasePos, WorkPos1 := #iA1UpClamp_WorkPos, BasePos2 := #iA2UpClamp_BasePos, WorkPos2 := #iA2UpClamp_WorkPos, Palette_on_station := #Pallet_On_Tippler, Hydraulic_unit_rdy := #Hydraulic_Ready.Q, MoveToWorkPos => #UpperClamps.MoveToWorkPos, MoveToBasePos => #UpperClamps.MoveToBasePos)
   END_RUNG
   RUNG wire#powerrail
      Contact( #Arms_clampsOperPos )
   END_RUNG wire#w2
   RUNG wire#powerrail
      Contact( #Arms_basePos )
      wire#w1
      { S7_Templates := "SrcType := Int" } EQ_Contact(in1 := #"Step", in2 := 0)
   END_RUNG wire#w2
   RUNG wire#powerrail
      I_Contact( #Pallet_On_Tippler )
   END_RUNG wire#w1
   RUNG wire#powerrail
      { S7_Templates := "SrcType := Int" } EQ_Contact(in1 := #"Step", in2 := 2)
   END_RUNG wire#w2
   // the same network as SCL:
   #UpperClamps(Req_arms_move_to_workPos := #ReqUpperClampsClose,   // "Clamp"
                Req_arms_move_to_basePos := #ReqUpperClampsOpen,
                BasePos1 := #iA1UpClamp_BasePos,
                WorkPos1 := #iA1UpClamp_WorkPos,
                BasePos2 := #iA2UpClamp_BasePos,
                WorkPos2 := #iA2UpClamp_WorkPos,
                Palette_on_station := #Pallet_On_Tippler,
                Arms_in_pos := #Arms_clampsOperPos OR ((#Arms_basePos OR NOT #Pallet_On_Tippler) AND (#"Step" = 0)) OR (#"Step" = 2),
                Hydraulic_unit_rdy := #Hydraulic_Ready.Q,
                MoveToWorkPos => #UpperClamps.MoveToWorkPos,
                MoveToBasePos => #UpperClamps.MoveToBasePos);
END_REGION

REGION Network 13
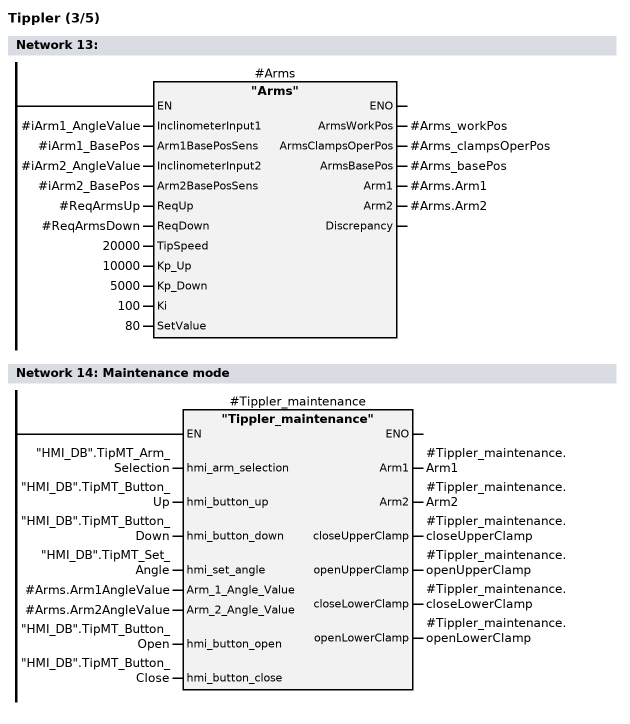
   RUNG wire#powerrail
      #Arms(InclinometerInput1 := #iArm1_AngleValue, Arm1BasePosSens := #iArm1_BasePos, InclinometerInput2 := #iArm2_AngleValue, Arm2BasePosSens := #iArm2_BasePos, ReqUp := #ReqArmsUp, ReqDown := #ReqArmsDown, TipSpeed := 20000, Kp_Up := 10000, Kp_Down := 5000, Ki := 100, SetValue := 80, ArmsWorkPos => #Arms_workPos, ArmsClampsOperPos => #Arms_clampsOperPos, ArmsBasePos => #Arms_basePos, Arm1 => #Arms.Arm1, Arm2 => #Arms.Arm2, Discrepancy =>)
   END_RUNG
   // the same network as SCL:
   #Arms(InclinometerInput1 := #iArm1_AngleValue,   // "Arms"
         Arm1BasePosSens := #iArm1_BasePos,
         InclinometerInput2 := #iArm2_AngleValue,
         Arm2BasePosSens := #iArm2_BasePos,
         ReqUp := #ReqArmsUp,
         ReqDown := #ReqArmsDown,
         TipSpeed := 20000,
         Kp_Up := 10000,
         Kp_Down := 5000,
         Ki := 100,
         SetValue := 80,
         ArmsWorkPos => #Arms_workPos,
         ArmsClampsOperPos => #Arms_clampsOperPos,
         ArmsBasePos => #Arms_basePos,
         Arm1 => #Arms.Arm1,
         Arm2 => #Arms.Arm2);
END_REGION

REGION Network 14: Maintenance mode
   RUNG wire#powerrail
      #Tippler_maintenance(hmi_arm_selection := "HMI_DB".TipMT_Arm_Selection, hmi_button_up := "HMI_DB".TipMT_Button_Up, hmi_button_down := "HMI_DB".TipMT_Button_Down, hmi_set_angle := "HMI_DB".TipMT_Set_Angle, Arm_1_Angle_Value := #Arms.Arm1AngleValue, Arm_2_Angle_Value := #Arms.Arm2AngleValue, hmi_button_open := "HMI_DB".TipMT_Button_Open, hmi_button_close := "HMI_DB".TipMT_Button_Close, Arm1 => #Tippler_maintenance.Arm1, Arm2 => #Tippler_maintenance.Arm2, closeUpperClamp => #Tippler_maintenance.closeUpperClamp, openUpperClamp => #Tippler_maintenance.openUpperClamp, closeLowerClamp => #Tippler_maintenance.closeLowerClamp, openLowerClamp => #Tippler_maintenance.openLowerClamp)
   END_RUNG
   // the same network as SCL:
   #Tippler_maintenance(hmi_arm_selection := "HMI_DB".TipMT_Arm_Selection,   // "Tippler_maintenance"
                        hmi_button_up := "HMI_DB".TipMT_Button_Up,
                        hmi_button_down := "HMI_DB".TipMT_Button_Down,
                        hmi_set_angle := "HMI_DB".TipMT_Set_Angle,
                        Arm_1_Angle_Value := #Arms.Arm1AngleValue,
                        Arm_2_Angle_Value := #Arms.Arm2AngleValue,
                        hmi_button_open := "HMI_DB".TipMT_Button_Open,
                        hmi_button_close := "HMI_DB".TipMT_Button_Close,
                        Arm1 => #Tippler_maintenance.Arm1,
                        Arm2 => #Tippler_maintenance.Arm2,
                        closeUpperClamp => #Tippler_maintenance.closeUpperClamp,
                        openUpperClamp => #Tippler_maintenance.openUpperClamp,
                        closeLowerClamp => #Tippler_maintenance.closeLowerClamp,
                        openLowerClamp => #Tippler_maintenance.openLowerClamp);
END_REGION

REGION Network 15: Arm Valves Control
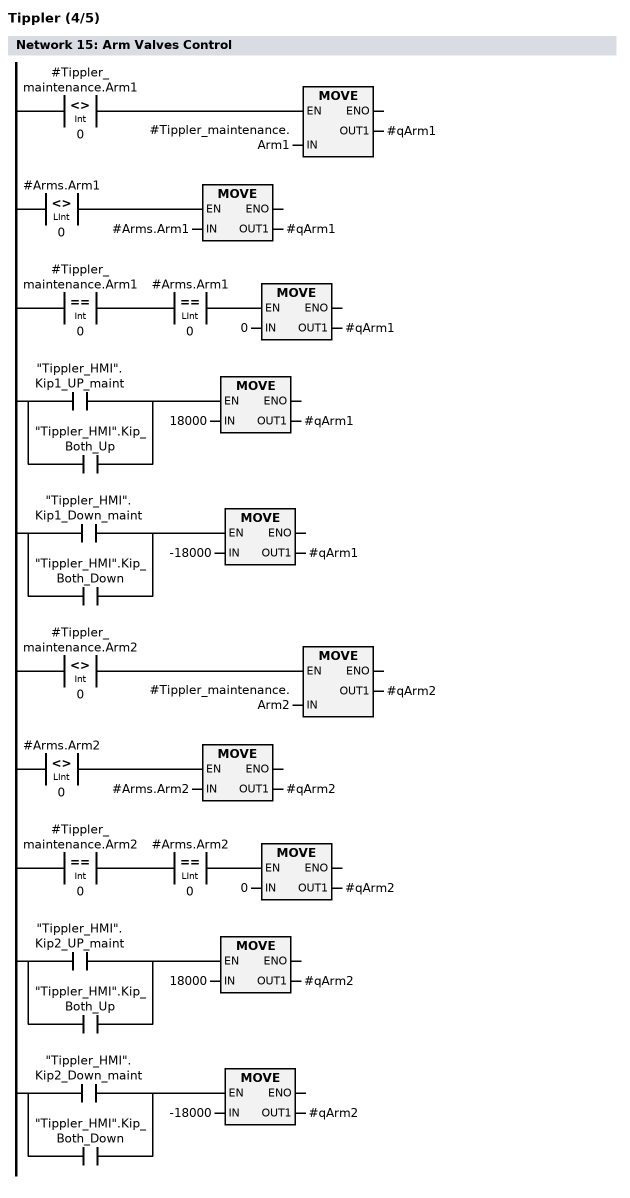
   RUNG wire#powerrail
      { S7_Templates := "SrcType := Int" } NE_Contact(in1 := #Tippler_maintenance.Arm1, in2 := 0)
      Move(in := #Tippler_maintenance.Arm1, out1 => #qArm1)
   END_RUNG
   RUNG wire#powerrail
      { S7_Templates := "SrcType := LInt" } NE_Contact(in1 := #Arms.Arm1, in2 := 0)
      Move(in := #Arms.Arm1, out1 => #qArm1)
   END_RUNG
   RUNG wire#powerrail
      { S7_Templates := "SrcType := Int" } EQ_Contact(in1 := #Tippler_maintenance.Arm1, in2 := 0)
      { S7_Templates := "SrcType := LInt" } EQ_Contact(in1 := #Arms.Arm1, in2 := 0)
      Move(in := 0, out1 => #qArm1)
   END_RUNG
   RUNG wire#powerrail
      Contact( "Tippler_HMI".Kip1_UP_maint )
      wire#w1
      Move(in := 18000, out1 => #qArm1)
   END_RUNG
   RUNG wire#powerrail
      Contact( "Tippler_HMI".Kip_Both_Up )
   END_RUNG wire#w1
   RUNG wire#powerrail
      Contact( "Tippler_HMI".Kip1_Down_maint )
      wire#w2
      Move(in := -18000, out1 => #qArm1)
   END_RUNG
   RUNG wire#powerrail
      Contact( "Tippler_HMI".Kip_Both_Down )
   END_RUNG wire#w2
   RUNG wire#powerrail
      { S7_Templates := "SrcType := Int" } NE_Contact(in1 := #Tippler_maintenance.Arm2, in2 := 0)
      Move(in := #Tippler_maintenance.Arm2, out1 => #qArm2)
   END_RUNG
   RUNG wire#powerrail
      { S7_Templates := "SrcType := LInt" } NE_Contact(in1 := #Arms.Arm2, in2 := 0)
      Move(in := #Arms.Arm2, out1 => #qArm2)
   END_RUNG
   RUNG wire#powerrail
      { S7_Templates := "SrcType := Int" } EQ_Contact(in1 := #Tippler_maintenance.Arm2, in2 := 0)
      { S7_Templates := "SrcType := LInt" } EQ_Contact(in1 := #Arms.Arm2, in2 := 0)
      Move(in := 0, out1 => #qArm2)
   END_RUNG
   RUNG wire#powerrail
      Contact( "Tippler_HMI".Kip2_UP_maint )
      wire#w3
      Move(in := 18000, out1 => #qArm2)
   END_RUNG
   RUNG wire#powerrail
      Contact( "Tippler_HMI".Kip_Both_Up )
   END_RUNG wire#w3
   RUNG wire#powerrail
      Contact( "Tippler_HMI".Kip2_Down_maint )
      wire#w4
      Move(in := -18000, out1 => #qArm2)
   END_RUNG
   RUNG wire#powerrail
      Contact( "Tippler_HMI".Kip_Both_Down )
   END_RUNG wire#w4
   // the same network as SCL:
   IF #Tippler_maintenance.Arm1 <> 0 THEN #qArm1 := #Tippler_maintenance.Arm1; END_IF;
   IF #Arms.Arm1 <> 0 THEN #qArm1 := #Arms.Arm1; END_IF;
   IF (#Tippler_maintenance.Arm1 = 0) AND (#Arms.Arm1 = 0) THEN #qArm1 := 0; END_IF;
   IF "Tippler_HMI".Kip1_UP_maint OR "Tippler_HMI".Kip_Both_Up THEN #qArm1 := 18000; END_IF;
   IF "Tippler_HMI".Kip1_Down_maint OR "Tippler_HMI".Kip_Both_Down THEN #qArm1 := -18000; END_IF;
   IF #Tippler_maintenance.Arm2 <> 0 THEN #qArm2 := #Tippler_maintenance.Arm2; END_IF;
   IF #Arms.Arm2 <> 0 THEN #qArm2 := #Arms.Arm2; END_IF;
   IF (#Tippler_maintenance.Arm2 = 0) AND (#Arms.Arm2 = 0) THEN #qArm2 := 0; END_IF;
   IF "Tippler_HMI".Kip2_UP_maint OR "Tippler_HMI".Kip_Both_Up THEN #qArm2 := 18000; END_IF;
   IF "Tippler_HMI".Kip2_Down_maint OR "Tippler_HMI".Kip_Both_Down THEN #qArm2 := -18000; END_IF;
END_REGION

REGION Network 16: Clamps Valve Control
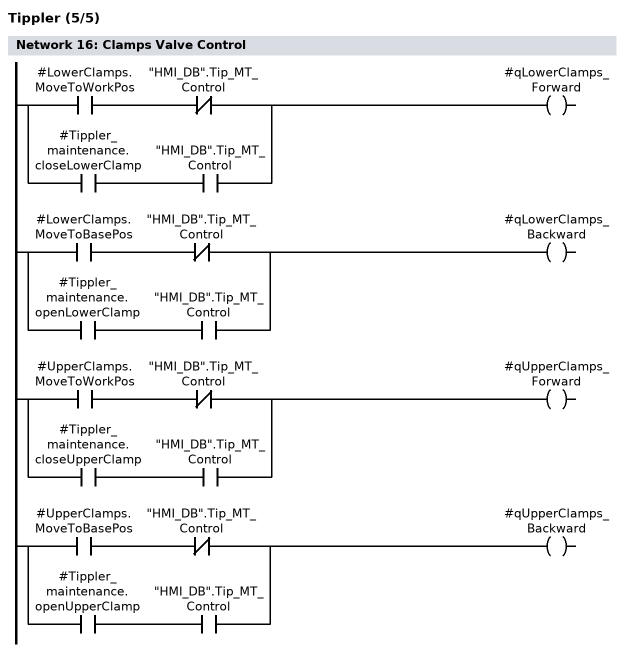
   RUNG wire#powerrail
      Contact( #LowerClamps.MoveToWorkPos )
      I_Contact( "HMI_DB".Tip_MT_Control )
      wire#w1
      Coil( #qLowerClamps_Forward )
   END_RUNG
   RUNG wire#powerrail
      Contact( #Tippler_maintenance.closeLowerClamp )
      Contact( "HMI_DB".Tip_MT_Control )
   END_RUNG wire#w1
   RUNG wire#powerrail
      Contact( #LowerClamps.MoveToBasePos )
      I_Contact( "HMI_DB".Tip_MT_Control )
      wire#w2
      Coil( #qLowerClamps_Backward )
   END_RUNG
   RUNG wire#powerrail
      Contact( #Tippler_maintenance.openLowerClamp )
      Contact( "HMI_DB".Tip_MT_Control )
   END_RUNG wire#w2
   RUNG wire#powerrail
      Contact( #UpperClamps.MoveToWorkPos )
      I_Contact( "HMI_DB".Tip_MT_Control )
      wire#w3
      Coil( #qUpperClamps_Forward )
   END_RUNG
   RUNG wire#powerrail
      Contact( #Tippler_maintenance.closeUpperClamp )
      Contact( "HMI_DB".Tip_MT_Control )
   END_RUNG wire#w3
   RUNG wire#powerrail
      Contact( #UpperClamps.MoveToBasePos )
      I_Contact( "HMI_DB".Tip_MT_Control )
      wire#w4
      Coil( #qUpperClamps_Backward )
   END_RUNG
   RUNG wire#powerrail
      Contact( #Tippler_maintenance.openUpperClamp )
      Contact( "HMI_DB".Tip_MT_Control )
   END_RUNG wire#w4
   // the same network as SCL:
   #qLowerClamps_Forward := (#LowerClamps.MoveToWorkPos AND NOT "HMI_DB".Tip_MT_Control) OR (#Tippler_maintenance.closeLowerClamp AND "HMI_DB".Tip_MT_Control);
   #qLowerClamps_Backward := (#LowerClamps.MoveToBasePos AND NOT "HMI_DB".Tip_MT_Control) OR (#Tippler_maintenance.openLowerClamp AND "HMI_DB".Tip_MT_Control);
   #qUpperClamps_Forward := (#UpperClamps.MoveToWorkPos AND NOT "HMI_DB".Tip_MT_Control) OR (#Tippler_maintenance.closeUpperClamp AND "HMI_DB".Tip_MT_Control);
   #qUpperClamps_Backward := (#UpperClamps.MoveToBasePos AND NOT "HMI_DB".Tip_MT_Control) OR (#Tippler_maintenance.openUpperClamp AND "HMI_DB".Tip_MT_Control);
END_REGION
END_FUNCTION_BLOCK

FUNCTION_BLOCK "Clamp"   // FB431, LAD
{ S7_Optimized_Access := 'TRUE' }
// stored: AutoNumber false, MemoryReserve 100, SetENOAutomatically false
   VAR_INPUT
      Req_arms_move_to_workPos : Bool;
      Req_arms_move_to_basePos : Bool;
      BasePos1 : Bool;
      WorkPos1 : Bool;
      BasePos2 : Bool;
      WorkPos2 : Bool;
      Palette_on_station : Bool;
      Arms_in_pos : Bool;
      Hydraulic_unit_rdy : Bool;
   END_VAR
   VAR_OUTPUT
      MoveToWorkPos : Bool;
      MoveToBasePos : Bool;
   END_VAR
   VAR
      Alarm_Clamp_Not_Close_Properly { S7_SetPoint := 'True'} : TON_TIME;
      Alarm_Clamp_Not_Open_Properly { S7_SetPoint := 'True'} : TON_TIME;
   END_VAR
BEGIN

REGION Network 1: Open Clamps
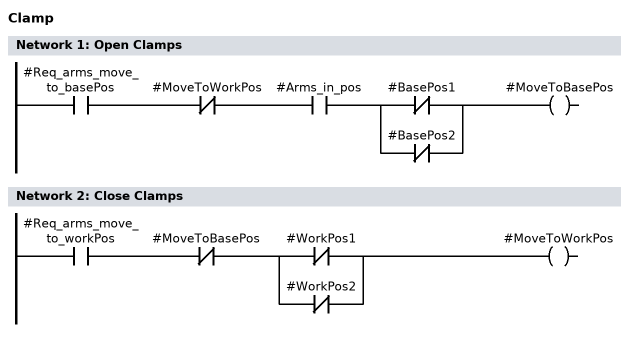
   RUNG wire#powerrail
      Contact( #Req_arms_move_to_basePos )
      I_Contact( #MoveToWorkPos )
      Contact( #Arms_in_pos )
      wire#w1
      I_Contact( #BasePos1 )
      wire#w2
      Coil( #MoveToBasePos )
   END_RUNG
   RUNG wire#w1
      I_Contact( #BasePos2 )
   END_RUNG wire#w2
   // the same network as SCL:
   #MoveToBasePos := #Req_arms_move_to_basePos AND NOT #MoveToWorkPos AND #Arms_in_pos AND (NOT #BasePos1 OR NOT #BasePos2);
END_REGION

REGION Network 2: Close Clamps
   RUNG wire#powerrail
      Contact( #Req_arms_move_to_workPos )
      I_Contact( #MoveToBasePos )
      wire#w1
      I_Contact( #WorkPos1 )
      wire#w2
      Coil( #MoveToWorkPos )
   END_RUNG
   RUNG wire#w1
      I_Contact( #WorkPos2 )
   END_RUNG wire#w2
   // the same network as SCL:
   #MoveToWorkPos := #Req_arms_move_to_workPos AND NOT #MoveToBasePos AND (NOT #WorkPos1 OR NOT #WorkPos2);
END_REGION

REGION Network 3 (SCL): Alarm Clamps not in position
   #Alarm_Clamp_Not_Close_Properly.TON(IN:=#MoveToWorkPos = 1 AND (#WorkPos1 = 0 OR #WorkPos2 = 0),
                                       PT:=T#3s);
   #Alarm_Clamp_Not_Open_Properly.TON(IN:=#MoveToBasePos = 1 AND (#BasePos1 = 0 OR #BasePos2 = 0) ,
                                       PT:=T#3s);
END_REGION
END_FUNCTION_BLOCK

FUNCTION_BLOCK "Arms"   // FB430, LAD
{ S7_Optimized_Access := 'TRUE' }
// stored: AutoNumber false, MemoryReserve 100, SetENOAutomatically false
   VAR_INPUT
      InclinometerInput1 : Int;
      Arm1BasePosSens : Bool;
      InclinometerInput2 : Int;
      Arm2BasePosSens : Bool;
      ReqUp : Bool;
      ReqDown : Bool;
      TipSpeed : Int := 15000;
      Kp_Up : Int := 100;
      Kp_Down : Int;
      Ki : Int;
      SetValue : Int := 78;
   END_VAR
   VAR_OUTPUT
      ArmsWorkPos : Bool;
      ArmsClampsOperPos : Bool;
      ArmsBasePos : Bool;
      Arm1 : Int;
      Arm2 : Int;
      Discrepancy : Real;   // absolut discrepancy value between arms
   END_VAR
   VAR
      Arm1AngleValue : Real;
      Arm2AngleValue : Real;
      Arm1BasePos : Bool;
      Arm2BasePos : Bool;
      Arm1WorkPos : Bool;
      Arm2WorkPos : Bool;
      Arm1ClampsOperPos : Bool;
      Arm2ClampsOperPos : Bool;
      Integral : Real;
      MAX_Output : Int := 7468;
      MIN_Output : Int := -7468;
      FilteredDiscrepancy : Real;
      Alpha : Real;
      TipSpeedDown : Int;
      SpeedRampTimerDown { S7_SetPoint := 'True'} : TON_TIME;
      SpeedRampTimerUP { S7_SetPoint := 'True'} : TON_TIME;
      TipSpeedAdjusted { S7_SetPoint := 'True'} : Int;
      SpeedReduction : Int := 3000;
      Delta : Int;
      PrevOutput : Int;
   END_VAR
   VAR_TEMP
      P_term : Int;
      I_term : Int;
      output : LInt;
      "dt" : Real;
      Var1 : Real;
   END_VAR
BEGIN

REGION Network 1: Scale Arm1
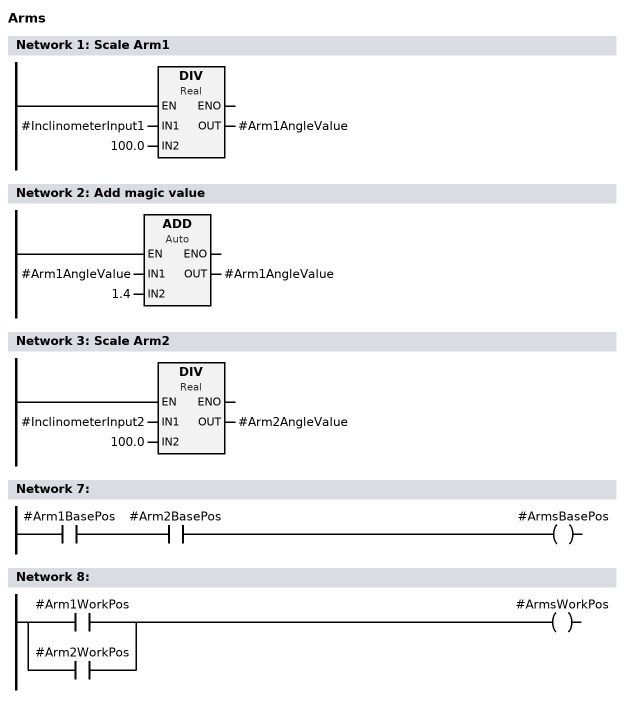
   RUNG wire#powerrail
      { S7_Templates := "SrcType := Real" } Div(in1 := #InclinometerInput1, in2 := 100.0, out => #Arm1AngleValue)
   END_RUNG
   // the same network as SCL:
   #Arm1AngleValue := #InclinometerInput1 / 100.0;
END_REGION

REGION Network 2: Add magic value
   RUNG wire#powerrail
      Add(in1 := #Arm1AngleValue, in2 := 1.4, out => #Arm1AngleValue)
   END_RUNG
   // the same network as SCL:
   #Arm1AngleValue := #Arm1AngleValue + 1.4;
END_REGION

REGION Network 3: Scale Arm2
   RUNG wire#powerrail
      { S7_Templates := "SrcType := Real" } Div(in1 := #InclinometerInput2, in2 := 100.0, out => #Arm2AngleValue)
   END_RUNG
   // the same network as SCL:
   #Arm2AngleValue := #InclinometerInput2 / 100.0;
END_REGION

REGION Network 4 (SCL): Base position Arm1 Arm2
   IF #Arm1AngleValue < 0.05 AND #Arm1BasePosSens THEN
       //BasePos arm 1 
       #Arm1BasePos := TRUE;
   ELSE
       #Arm1BasePos := FALSE;
   END_IF;

   IF #Arm2AngleValue < 0.15 AND #Arm2BasePosSens THEN
       //BasePos arm 2 
       #Arm2BasePos := TRUE;
   ELSE
       #Arm2BasePos := FALSE;
   END_IF;
END_REGION

REGION Network 5 (SCL): Clamps operating position
   #ArmsClampsOperPos := 0;
   IF #Arm1AngleValue > 2 AND #Arm1AngleValue < 3.5 THEN
       //BasePos arm 1 
       #Arm1ClampsOperPos := TRUE;
   ELSE
       #Arm1ClampsOperPos := FALSE;
   END_IF;

   IF #Arm2AngleValue > 2 AND #Arm2AngleValue < 3.5 THEN
       //BasePos arm 2 
       #Arm2ClampsOperPos := TRUE;
   ELSE
       #Arm2ClampsOperPos := FALSE;
   END_IF;

   IF (#Arm1ClampsOperPos OR #Arm2ClampsOperPos) AND ABS(#Discrepancy) < 1.2 THEN
       #ArmsClampsOperPos := 1;
   END_IF;
END_REGION

REGION Network 6 (SCL): Work position Arm1 Arm2
   IF ABS(#Arm1AngleValue - #SetValue) < 1 THEN
       //WorkPos arm 1 
        #Arm1WorkPos := TRUE;
   ELSE
       #Arm1WorkPos := FALSE;
   END_IF;
   IF ABS(#Arm2AngleValue - #SetValue) < 1  THEN
       //WorkPos arm 2 
       #Arm2WorkPos := TRUE;
   ELSE
       #Arm2WorkPos := FALSE;
   END_IF;
END_REGION

REGION Network 7
   RUNG wire#powerrail
      Contact( #Arm1BasePos )
      Contact( #Arm2BasePos )
      Coil( #ArmsBasePos )
   END_RUNG
   // the same network as SCL:
   #ArmsBasePos := #Arm1BasePos AND #Arm2BasePos;
END_REGION

REGION Network 8
   RUNG wire#powerrail
      Contact( #Arm1WorkPos )
      wire#w1
      Coil( #ArmsWorkPos )
   END_RUNG
   RUNG wire#powerrail
      Contact( #Arm2WorkPos )
   END_RUNG wire#w1
   // the same network as SCL:
   #ArmsWorkPos := #Arm1WorkPos OR #Arm2WorkPos;
END_REGION

REGION Network 9 (SCL): discrepancy value between arms
   // -  Arm1 is lower
   // + Arm 1 is higher
   #Discrepancy := #Arm1AngleValue - #Arm2AngleValue;
END_REGION

REGION Network 10 (SCL): MoveArms to workPos by ButtonUp
   // Reset prędkości
   #Arm1 := 0;
   #Arm2 := 0;
   #dt := 0.02; // Czas próbkowania np. 20ms
   #Integral := 0.0;
   #MAX_Output := 3500;
   #MIN_Output := -3500;
   #output := 0;

   // Filtrowanie sygnału z inklinometru (prosty filtr IIR)
   // 

   #SpeedRampTimerUP(IN:= #ReqUp AND "Tippler_DB".Hydraulic_Ready.Q,
                   PT:=T#10s); //4
   IF NOT #SpeedRampTimerUP.Q AND #ReqUp THEN
       #Var1 := INT_TO_REAL(TIME_TO_INT(#SpeedRampTimerUP.ET)) / INT_TO_REAL(TIME_TO_INT(#SpeedRampTimerUP.PT));

       #TipSpeed := 10500 + #Var1 * 9500; //13000 5000
   ELSIF #Arm1AngleValue >= 70.0 THEN
       #TipSpeed := 14500 + 5500 * (81 - #Arm1AngleValue) / 11;
   END_IF;


   #SpeedRampTimerDown(IN := #ReqDown AND "Tippler_DB".Hydraulic_Ready.Q,
                   PT := T#10s); //4
   IF NOT #SpeedRampTimerDown.Q AND #ReqDown THEN
       #Var1 := INT_TO_REAL(TIME_TO_INT(#SpeedRampTimerDown.ET)) / INT_TO_REAL(TIME_TO_INT(#SpeedRampTimerDown.PT));

       #TipSpeed := 10000 + #Var1 * 8000; //10300 7700

   ELSIF #SpeedRampTimerDown.Q AND #ReqDown THEN
       #TipSpeed := 18000;
       IF #Arm1AngleValue <= 7.0 THEN
           #TipSpeed := 10500 + 7500 * (#Arm1AngleValue / 7);
       END_IF;

   END_IF;



   // Jazda w górę
   IF #ReqUp THEN
       #Alpha := 0.05; // tłumienie (0.05 - 0.2 zalecane)
       #FilteredDiscrepancy := #FilteredDiscrepancy + #Alpha * (#Discrepancy - #FilteredDiscrepancy);


       // Arm1: master – jedzie niezależnie do pozycji roboczej
       IF NOT #Arm1WorkPos THEN
           #Arm1 :=#TipSpeed -0;
       END_IF;

       // Arm2: slave – jedzie niezależnie, ale korygowany względem Arm1
       IF NOT #Arm2WorkPos THEN
           // Człon P
           IF NOT "Arm1_UpperClampClosed" THEN
               #Kp_Up := 300;
           END_IF;
           #P_term := REAL_TO_INT(#FilteredDiscrepancy * #Kp_Up);

           // Ograniczenie
           IF #P_term > #MAX_Output THEN
               #output := #MAX_Output;
           ELSIF #P_term < #MIN_Output THEN
               #output := #MIN_Output;
           ELSE
               #output := #P_term;
           END_IF;

           #Delta := #output - #PrevOutput;

           IF #Delta > 10 THEN
               #output := #PrevOutput + 10;
           ELSIF #Delta < -10 THEN
               #output := #PrevOutput - 10;
           END_IF;

           // Zapisz bieżący output jako poprzedni na następny cykl
           #PrevOutput := #output;

           #Arm2 := #Arm1 + #output - 1000;
       END_IF;

       // Jazda w dół
   ELSIF #ReqDown THEN
       #Alpha := 0.02; // tłumienie (0.05 - 0.2 zalecane) //im mniejsze tym bardziej ujednolica
       #FilteredDiscrepancy := #FilteredDiscrepancy + #Alpha * (#Discrepancy - #FilteredDiscrepancy);


       // Arm1: master – jedzie niezależnie do pozycji bazowej
       IF NOT #Arm1BasePos THEN
           IF #Arm1AngleValue > 60 THEN
               #TipSpeedDown := #TipSpeed;
           ELSE
               #TipSpeedDown := #TipSpeed;
           END_IF;
           #Arm1 := - #TipSpeedDown +0;
       END_IF;

       // Arm2: slave – jedzie niezależnie, korygowany względem Arm1
       IF NOT #Arm2BasePos THEN
           #MAX_Output := 3000;
           #MIN_Output := -3000;

           // Człon P
           #P_term := REAL_TO_INT(#FilteredDiscrepancy * #Kp_Down);

           // Ograniczenie
           IF #P_term > #MAX_Output THEN
               #output := #MAX_Output;
           ELSIF #P_term < #MIN_Output THEN
               #output := #MIN_Output;
           ELSE
               #output := #P_term;
           END_IF;

           // Ograniczenie skoku wartości output względem poprzedniego cyklu
           #Delta := #output - #PrevOutput;

           IF #Delta > 4 THEN
               #output := #PrevOutput + 4;
           ELSIF #Delta < -4 THEN
               #output := #PrevOutput - 4;
           END_IF;

           // Zapisz bieżący output jako poprzedni na następny cykl
           #PrevOutput := #output;

           #Arm2 := #Arm1 + #output + 900;
       END_IF;

   END_IF;
END_REGION
END_FUNCTION_BLOCK

FUNCTION_BLOCK "Tippler_maintenance"   // FB401, LAD
{ S7_Optimized_Access := 'TRUE' }
// stored: AutoNumber false, MemoryReserve 100, SetENOAutomatically false
   VAR_INPUT
      hmi_arm_selection : Int;
      hmi_button_up : Bool;
      hmi_button_down : Bool;
      hmi_set_angle : Int;
      Arm_1_Angle_Value : Real;
      Arm_2_Angle_Value : Real;
      hmi_button_open : Bool;
      hmi_button_close : Bool;
   END_VAR
   VAR_OUTPUT
      Arm1 : Int;
      Arm2 : Int;
      closeUpperClamp : Bool;
      openUpperClamp : Bool;
      closeLowerClamp : Bool;
      openLowerClamp : Bool;
   END_VAR
   VAR
      Arm1SetPosReached : Bool;
      Arm2SetPosReached : Bool;
      speed : Int;
   END_VAR
BEGIN

REGION Network 1 (SCL): Manual operating
   #Arm1 := 0;
   #Arm2 := 0;
   #speed := 0;
   IF #Arm_1_Angle_Value > 50 OR #Arm_2_Angle_Value > 50 THEN
       #speed := 15000;
   ELSE
       #speed := 20000;
   END_IF;
   IF #hmi_arm_selection = 1 THEN
       IF #hmi_button_up AND #hmi_set_angle > #Arm_1_Angle_Value THEN
           #Arm1 :=#speed;
           #Arm2 := 0;
           #closeUpperClamp := FALSE;
           #closeLowerClamp := FALSE;
           #openUpperClamp := FALSE;
           #openLowerClamp := FALSE;
       ELSIF #hmi_button_down THEN
           #Arm1 := -#speed;
           #Arm2 := 0;
           #closeUpperClamp := FALSE;
           #closeLowerClamp := FALSE;
           #openUpperClamp := FALSE;
           #openLowerClamp := FALSE;
       ELSIF #hmi_button_close THEN
           #Arm1 := 0;
           #Arm2 := 0;
           #closeUpperClamp := TRUE;
           #closeLowerClamp := FALSE;
           #openUpperClamp := FALSE; 
           #openLowerClamp := FALSE;
       ELSIF #hmi_button_open THEN
           #Arm1 := 0;
           #Arm2 := 0;
           #closeUpperClamp := FALSE;
           #closeLowerClamp := FALSE;
           #openUpperClamp := TRUE;
           #openLowerClamp := FALSE;
       ELSE
           #Arm1 := 0;
           #Arm2 := 0;
           #closeUpperClamp := FALSE;
           #closeLowerClamp := FALSE;
           #openUpperClamp := FALSE;
           #openLowerClamp := FALSE;
       END_IF;
   ELSIF #hmi_arm_selection = 2  THEN
       IF #hmi_button_up AND #hmi_set_angle > #Arm_2_Angle_Value THEN
           #Arm2 := #speed;
           #Arm1 := 0;
           #closeUpperClamp := FALSE;
           #closeLowerClamp := FALSE;
           #openUpperClamp := FALSE;
           #openLowerClamp := FALSE;
       ELSIF #hmi_button_down THEN
           #Arm2 := -#speed;
           #Arm1 := 0;
           #closeUpperClamp := FALSE;
           #closeLowerClamp := FALSE;
           #openUpperClamp := FALSE;
           #openLowerClamp := FALSE;
       ELSIF #hmi_button_close THEN
           #Arm1 := 0;
           #Arm2 := 0;
           #closeUpperClamp := FALSE;
           #closeLowerClamp := TRUE;
           #openUpperClamp := FALSE;
           #openLowerClamp := FALSE;
       ELSIF #hmi_button_open THEN
           #Arm1 := 0;
           #Arm2 := 0;
           #closeUpperClamp := FALSE;
           #closeLowerClamp := FALSE;
           #openUpperClamp := FALSE;
           #openLowerClamp := TRUE;
       ELSE
           #Arm2 := 0;
           #Arm1 := 0;
           #closeUpperClamp := FALSE;
           #closeLowerClamp := FALSE;
           #openUpperClamp := FALSE;
           #openLowerClamp := FALSE;
       END_IF;
   ELSIF #hmi_arm_selection = 0 THEN
       IF #hmi_button_up THEN
           IF #hmi_set_angle > #Arm_2_Angle_Value AND #hmi_set_angle > #Arm_1_Angle_Value THEN
               #Arm1 := #speed;
               #Arm2 := #speed;
               #closeUpperClamp := FALSE;
               #closeLowerClamp := FALSE;
               #openUpperClamp := FALSE;
               #openLowerClamp := FALSE;
           ELSIF #hmi_set_angle > #Arm_2_Angle_Value AND #hmi_set_angle < #Arm_1_Angle_Value THEN
               #Arm1 := 0;
               #Arm2 := #speed;
               #closeUpperClamp := FALSE;
               #closeLowerClamp := FALSE;
               #openUpperClamp := FALSE;
               #openLowerClamp := FALSE;
           ELSIF #hmi_set_angle < #Arm_2_Angle_Value AND #hmi_set_angle > #Arm_1_Angle_Value THEN
               #Arm1 := #speed;
               #Arm2 := 0;
               #closeUpperClamp := FALSE;
               #closeLowerClamp := FALSE;
               #openUpperClamp := FALSE;
               #openLowerClamp := FALSE;
           ELSE
               #Arm1 := 0;
               #Arm2 := 0;
               #closeUpperClamp := FALSE;
               #closeLowerClamp := FALSE;
               #openUpperClamp := FALSE;
               #openLowerClamp := FALSE;
           END_IF;
       ELSIF #hmi_button_down THEN
           #Arm2 := -#speed;
           #Arm1 := -#speed;
           #closeUpperClamp := FALSE;
           #closeLowerClamp := FALSE;
           #openUpperClamp := FALSE;
           #openLowerClamp := FALSE;
       ELSIF #hmi_button_close THEN
           #Arm1 := 0;
           #Arm2 := 0;
           #closeUpperClamp := TRUE;
           #closeLowerClamp := TRUE;
           #openUpperClamp := FALSE;
           #openLowerClamp := FALSE;
       ELSIF #hmi_button_open THEN
           #Arm1 := 0;
           #Arm2 := 0;
           #closeUpperClamp := FALSE;
           #closeLowerClamp := FALSE;
           #openUpperClamp := TRUE;
           #openLowerClamp := TRUE;
       ELSE
           #Arm2 := 0;
           #Arm1 := 0;
           #closeUpperClamp := FALSE;
           #closeLowerClamp := FALSE;
           #openUpperClamp := FALSE;
           #openLowerClamp := FALSE;
       END_IF;
   ELSE
       #Arm1 := 0;
       #Arm2 := 0;
       #closeUpperClamp := FALSE;
       #closeLowerClamp := FALSE;
       #openUpperClamp := FALSE;
       #openLowerClamp := FALSE;
   END_IF;
END_REGION

REGION Network 2 (SCL)
   IF #Arm_1_Angle_Value > #hmi_set_angle THEN
       #Arm1SetPosReached := 1;

   ELSE
       #Arm1SetPosReached := 0;
   END_IF;
   IF #Arm_2_Angle_Value > #hmi_set_angle THEN
       #Arm2SetPosReached := 1;
   ELSE
       #Arm2SetPosReached := 0;
   END_IF;
END_REGION
END_FUNCTION_BLOCK

ORGANIZATION_BLOCK "MC_PreServo"   // OB67, LAD, PreServo
{ S7_Optimized_Access := 'TRUE' }
// stored: SetENOAutomatically false
   VAR_INPUT
      Initial_Call : Bool;
      PIP_Input : Bool;
      PIP_Output : Bool;
      IO_System : USInt;
      Event_Count : Int;
      Synchronous : Bool;
      CycleTime : UDInt;
   END_VAR
BEGIN

REGION Network 1
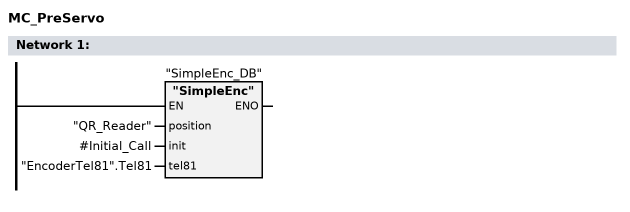
   RUNG wire#powerrail
      "SimpleEnc_DB"(position := "QR_Reader", init := #Initial_Call, tel81 := "EncoderTel81".Tel81)
   END_RUNG
   // the same network as SCL:
   "SimpleEnc_DB"(position := "QR_Reader", init := #Initial_Call, tel81 := "EncoderTel81".Tel81);   // "SimpleEnc"
END_REGION
END_ORGANIZATION_BLOCK

FUNCTION_BLOCK "SimpleEnc"
{ S7_Optimized_Access := 'FALSE' }
VERSION : 0.1
   VAR_INPUT 
      position : DInt;
      init : Bool;
   END_VAR

   VAR_IN_OUT 
      tel81 {InstructionName := 'PD_TEL81'; LibVersion := '7.0'} : PD_TEL81;
   END_VAR

   VAR 
      statError : Bool;
      statOldPos : DInt;
   END_VAR

   VAR_TEMP 
      tempReqCmd : Bool;
      tempDPos : DInt;
   END_VAR


BEGIN
	//=============================================================================
	// SIEMENS AG - zmodyfikowane dla pozycji w mm
	//-----------------------------------------------------------------------------
	// Functionality: make the encoder telegram 81 with position in mm
	//-----------------------------------------------------------------------------
	
	// Inicjalizacja
	IF #init THEN
	    #statOldPos := #position;                 // zapamiętaj startową pozycję w mm
	    #tel81.Input.G1_XIST1 := 0;               // wyzeruj inkrementalną
	    #tel81.Input.G1_XIST2 := DINT_TO_DWORD(#position);  // ustaw absolutną
	    #tel81.Input.G1_ZSW.SensorError := FALSE;
	    #statError := FALSE;
	END_IF;
	
	// Oblicz przyrost względem poprzedniej pozycji
	#tempDPos := #position - #statOldPos;
	
	// Zapisz przyrost (inkrementalna pozycja)
	#tel81.Input.G1_XIST1 := #tel81.Input.G1_XIST1 + DINT_TO_DWORD(#tempDPos);
	
	// Aktualizacja poprzedniej pozycji
	#statOldPos := #position;
	
	// Zapisz absolutną pozycję w mm
	#tel81.Input.G1_XIST2 := DINT_TO_DWORD(#position);
	#tel81.Input.G1_ZSW.AbsoluteValueCyclicallyExecuted := TRUE;
	
	// Obsługa błędu – uproszczona
	IF #statError THEN
	    IF #tel81.Output.G1_STW.AcknowledgeError THEN
	        #statError := FALSE;
	        #tel81.Input.G1_XIST1 := 0;
	        #tel81.Input.G1_XIST2 := DINT_TO_DWORD(#position);
	        #tel81.Input.G1_ZSW.SensorError := FALSE;
	    END_IF;
	END_IF;
	
	// Interpretuje żądania sterownika (STW)
	#tempReqCmd := #tel81.Output.G1_STW.Command0Request
	OR #tel81.Output.G1_STW.Command1Request
	OR #tel81.Output.G1_STW.Command2Request
	OR #tel81.Output.G1_STW.RequestParkingEncoder;
	
	// jeśli encoder jest tylko „mm” (brak obsługi innych trybów), traktujemy to jako błąd
	IF #tempReqCmd THEN
	    #tel81.Input.G1_ZSW.SensorError := TRUE;
	    #tel81.Input.G1_XIST2 := 16#0F01;
	    #statError := TRUE;
	END_IF;
	
END_FUNCTION_BLOCK

FUNCTION_BLOCK "Pallets_Transport_System"   // FB9, LAD
{ S7_Optimized_Access := 'TRUE' }
// stored: MemoryReserve 100, SetENOAutomatically false
   VAR
      NumberOfPallet { S7_SetPoint := 'True'} : Int;
      Map : Array[1..4, 1..12] of Bool;
      MoveDirection : Int;   // 1-L, 2-Up, 3-R, 4-Down
      FoundSelectedPallet : Bool;
      CanMove : Bool;
      Station_Next_Position : Array[1..2] of Int;
      SelectedPalletFound : Bool;
   END_VAR
   VAR_TEMP
      i : Int;
      j : Int;
      k : Int;
   END_VAR
BEGIN

REGION Network 1 (SCL)
   // Sprawdzenie, które elementy sa wybrane i nadanie im nowej pozycji
   #SelectedPalletFound := FALSE;

   FOR #k := 1 TO 24 DO
       IF "Pallets_Stations".Pallets[#k].IsSelected THEN
           #SelectedPalletFound := TRUE;
           EXIT;
       END_IF;
   END_FOR;

   IF #SelectedPalletFound THEN
       #Station_Next_Position := "Pallets_Stations".Pallets[#k].Station_Current_Position;

               CASE #MoveDirection OF
                   1:
                       IF #Station_Next_Position[2] > 1 THEN  // Check Left
                           #Station_Next_Position[2] := #Station_Next_Position[2] - 1;
                       ELSE
                           #CanMove := FALSE;
                       END_IF;
                   3:
                       IF (#Station_Next_Position[2] < 12) AND // Check Right
                           ((#Station_Next_Position[1] = 2 AND #Station_Next_Position[2] < 12) OR (#Station_Next_Position[1] <> 2 AND #Station_Next_Position[2] < 11)) THEN
                           #Station_Next_Position[2] := #Station_Next_Position[2] + 1;
                       ELSE
                           #CanMove := FALSE; 
                       END_IF;
                   2:
                       IF (#Station_Next_Position[2] = 1) OR
                           ((#Station_Next_Position[1] = 1 AND #Station_Next_Position[2] = 11) OR
                           (#Station_Next_Position[1] = 2 AND #Station_Next_Position[2] = 12) OR
                           (#Station_Next_Position[1] = 3 AND #Station_Next_Position[2] = 11) OR
                           (#Station_Next_Position[1] = 4 AND #Station_Next_Position[2] = 11)) THEN
                           IF #Station_Next_Position[1] > 1 THEN
                               // Ruch w ostatniej kolumnie
                               IF #Station_Next_Position[1] = 2 AND #Station_Next_Position[2] = 12 THEN
                                   #Station_Next_Position[1] := 1;
                                   #Station_Next_Position[2] := 11;
                               ELSE
                                   #Station_Next_Position[1] := #Station_Next_Position[1] - 1;
                               END_IF;
                           ELSE
                               #CanMove := FALSE;
                           END_IF;
                       ELSE
                           #CanMove := FALSE;
                       END_IF;
                   4:
                       IF (#Station_Next_Position[2] = 1) OR
                           ((#Station_Next_Position[1] = 1 AND #Station_Next_Position[2] = 11) OR
                           (#Station_Next_Position[1] = 2 AND #Station_Next_Position[2] = 12) OR
                           (#Station_Next_Position[1] = 3 AND #Station_Next_Position[2] = 11) OR
                           (#Station_Next_Position[1] = 4 AND #Station_Next_Position[2] = 11)) THEN
                           IF #Station_Next_Position[1] < 4 THEN
                               // Ruch w ostatniej kolumnie
                               IF #Station_Next_Position[1] = 1 AND #Station_Next_Position[2] = 11 THEN
                                   #Station_Next_Position[1] := 2;
                                   #Station_Next_Position[2] := 12;
                               ELSE
                                   #Station_Next_Position[1] := #Station_Next_Position[1] + 1;
                               END_IF;
                           ELSE
                               #CanMove := FALSE;
                           END_IF;
                       ELSE
                           #CanMove := FALSE;
                       END_IF;
               END_CASE;

               "Pallets_Stations".Pallets[#k].Station_Current_Position := #Station_Next_Position;

           ELSE
               #CanMove := FALSE; // żaden pallet nie był wybrany
           END_IF;
END_REGION
END_FUNCTION_BLOCK

FUNCTION "SQL" : Void   // FC2, LAD
{ S7_Optimized_Access := 'TRUE' }
// stored: SetENOAutomatically false
   VAR_TEMP
      tempDataReceived : Bool;   // temp flag for 'dataReceived' from FB 'LSql_Microsoft'
      tempAnalyzeDone : Bool;   // temp flag for 'done' from FB 'AnalyzeTokens'
      tempMetaDataAndRowsAvailable : Bool;   // temp flag for 'metaDataAndRowsAvailable' from FB 'AnalyzeTokens'
   END_VAR
BEGIN

REGION Network 1: TDS Connection and Communication Handling
   // this network handles the TDS connection and communication
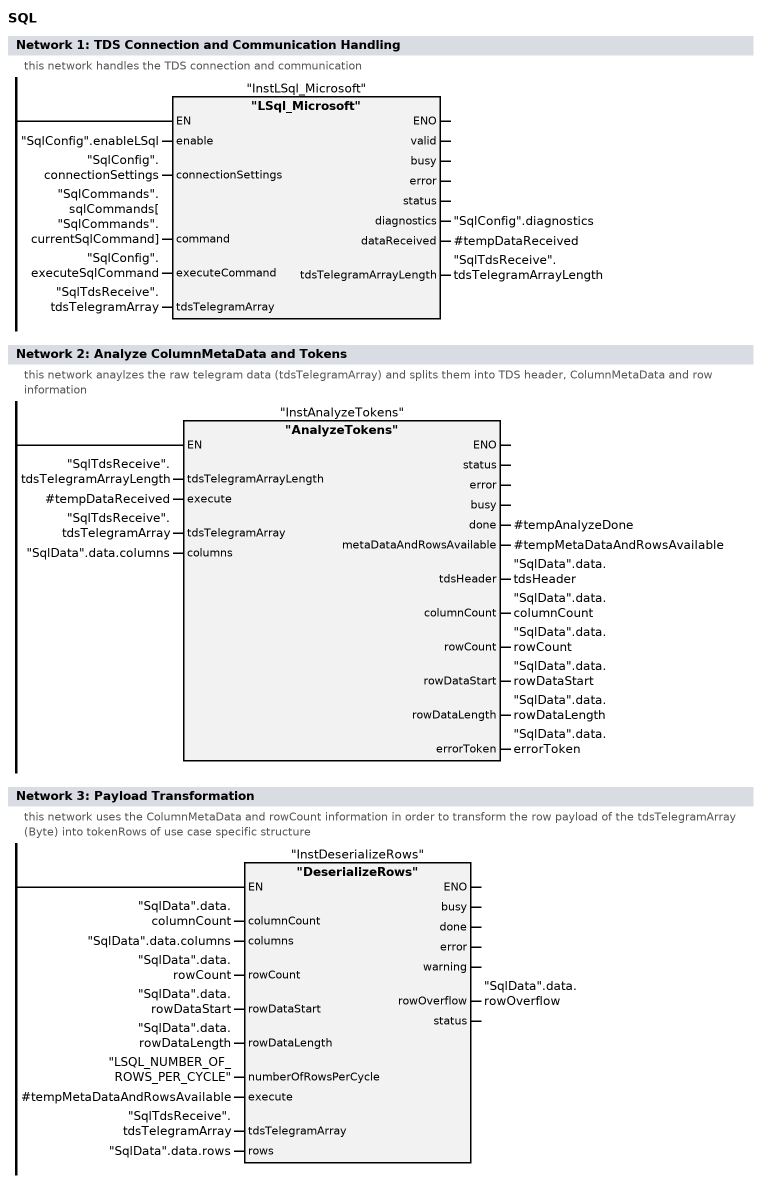
   RUNG wire#powerrail
      "InstLSql_Microsoft"(enable := "SqlConfig".enableLSql, connectionSettings := "SqlConfig".connectionSettings, command := "SqlCommands".sqlCommands["SqlCommands".currentSqlCommand], executeCommand := "SqlConfig".executeSqlCommand, tdsTelegramArray := "SqlTdsReceive".tdsTelegramArray, valid =>, busy =>, error =>, status =>, diagnostics => "SqlConfig".diagnostics, dataReceived => #tempDataReceived, tdsTelegramArrayLength => "SqlTdsReceive".tdsTelegramArrayLength)
   END_RUNG
   // the same network as SCL:
   "InstLSql_Microsoft"(enable := "SqlConfig".enableLSql,   // "LSql_Microsoft"
                        connectionSettings := "SqlConfig".connectionSettings,
                        command := "SqlCommands".sqlCommands["SqlCommands".currentSqlCommand],
                        executeCommand := "SqlConfig".executeSqlCommand,
                        tdsTelegramArray := "SqlTdsReceive".tdsTelegramArray,
                        diagnostics => "SqlConfig".diagnostics,
                        dataReceived => #tempDataReceived,
                        tdsTelegramArrayLength => "SqlTdsReceive".tdsTelegramArrayLength);
END_REGION

REGION Network 2: Analyze ColumnMetaData and Tokens
   // this network anaylzes the raw telegram data (tdsTelegramArray) and splits them into TDS header, ColumnMetaData and row information
   RUNG wire#powerrail
      "InstAnalyzeTokens"(tdsTelegramArrayLength := "SqlTdsReceive".tdsTelegramArrayLength, execute := #tempDataReceived, tdsTelegramArray := "SqlTdsReceive".tdsTelegramArray, columns := "SqlData".data.columns, status =>, error =>, busy =>, done => #tempAnalyzeDone, metaDataAndRowsAvailable => #tempMetaDataAndRowsAvailable, tdsHeader => "SqlData".data.tdsHeader, columnCount => "SqlData".data.columnCount, rowCount => "SqlData".data.rowCount, rowDataStart => "SqlData".data.rowDataStart, rowDataLength => "SqlData".data.rowDataLength, errorToken => "SqlData".data.errorToken)
   END_RUNG
   // the same network as SCL:
   "InstAnalyzeTokens"(tdsTelegramArrayLength := "SqlTdsReceive".tdsTelegramArrayLength,   // "AnalyzeTokens"
                       execute := #tempDataReceived,
                       tdsTelegramArray := "SqlTdsReceive".tdsTelegramArray,
                       columns := "SqlData".data.columns,
                       done => #tempAnalyzeDone,
                       metaDataAndRowsAvailable => #tempMetaDataAndRowsAvailable,
                       tdsHeader => "SqlData".data.tdsHeader,
                       columnCount => "SqlData".data.columnCount,
                       rowCount => "SqlData".data.rowCount,
                       rowDataStart => "SqlData".data.rowDataStart,
                       rowDataLength => "SqlData".data.rowDataLength,
                       errorToken => "SqlData".data.errorToken);
END_REGION

REGION Network 3: Payload Transformation
   // this network uses the ColumnMetaData and rowCount information in order to transform the row payload of the tdsTelegramArray (Byte) into tokenRows of use case specific structure
   RUNG wire#powerrail
      "InstDeserializeRows"(columnCount := "SqlData".data.columnCount, columns := "SqlData".data.columns, rowCount := "SqlData".data.rowCount, rowDataStart := "SqlData".data.rowDataStart, rowDataLength := "SqlData".data.rowDataLength, numberOfRowsPerCycle := "LSQL_NUMBER_OF_ROWS_PER_CYCLE", execute := #tempMetaDataAndRowsAvailable, tdsTelegramArray := "SqlTdsReceive".tdsTelegramArray, rows := "SqlData".data.rows, busy =>, done =>, error =>, warning =>, rowOverflow => "SqlData".data.rowOverflow, status =>)
   END_RUNG
   // the same network as SCL:
   "InstDeserializeRows"(columnCount := "SqlData".data.columnCount,   // "DeserializeRows"
                         columns := "SqlData".data.columns,
                         rowCount := "SqlData".data.rowCount,
                         rowDataStart := "SqlData".data.rowDataStart,
                         rowDataLength := "SqlData".data.rowDataLength,
                         numberOfRowsPerCycle := "LSQL_NUMBER_OF_ROWS_PER_CYCLE",
                         execute := #tempMetaDataAndRowsAvailable,
                         tdsTelegramArray := "SqlTdsReceive".tdsTelegramArray,
                         rows := "SqlData".data.rows,
                         rowOverflow => "SqlData".data.rowOverflow);
END_REGION
END_FUNCTION

FUNCTION_BLOCK "AnalyzeTokens"
TITLE = AnalyzeData
{ S7_Optimized_Access := 'TRUE' }
AUTHOR : 'SIEMENS AG'
VERSION : 3.0
//FB for analyzing raw SELECT batch data from Tabular Data Stream (tdsTelegramArray). It splits them into TDS header and Tokens, especially ColumnMetaData and Error token information. Output parameter also contain the number of received rows and their start and length in tdsTelegramArray
   VAR_INPUT 
      tdsTelegramArrayLength { ExternalAccessible := 'False'; ExternalVisible := 'False'; ExternalWritable := 'False'} : UDInt;   // number of bytes received by TDS
      execute { ExternalAccessible := 'False'; ExternalVisible := 'False'; ExternalWritable := 'False'} : Bool;   // bit flag for FB execution
   END_VAR

   VAR_OUTPUT 
      status { ExternalAccessible := 'False'; ExternalVisible := 'False'; ExternalWritable := 'False'} : Word := 16#0;   // output status code
      error { ExternalAccessible := 'False'; ExternalVisible := 'False'; ExternalWritable := 'False'} : Bool := FALSE;   // output error bit
      busy { ExternalAccessible := 'False'; ExternalVisible := 'False'; ExternalWritable := 'False'} : Bool := FALSE;   // output gor busy state
      done { ExternalAccessible := 'False'; ExternalVisible := 'False'; ExternalWritable := 'False'} : Bool := FALSE;   // flag for successful execution
      metaDataAndRowsAvailable { ExternalAccessible := 'False'; ExternalVisible := 'False'; ExternalWritable := 'False'} : Bool;   // flag for successful execution AND data contain ColumnMetaData and Rows
      tdsHeader { ExternalAccessible := 'False'; ExternalVisible := 'False'; ExternalWritable := 'False'} : "LSql_typePacketHeader";
      columnCount { ExternalAccessible := 'False'; ExternalVisible := 'False'; ExternalWritable := 'False'} : UInt := 0;   // number of columns
      rowCount { ExternalAccessible := 'False'; ExternalVisible := 'False'; ExternalWritable := 'False'} : UDInt := 0;   // number of rows
      rowDataStart { ExternalAccessible := 'False'; ExternalVisible := 'False'; ExternalWritable := 'False'} : UInt := 0;   // start byte address of row data area
      rowDataLength { ExternalAccessible := 'False'; ExternalVisible := 'False'; ExternalWritable := 'False'} : UDInt := 0;   // byte length of row data area
      errorToken { ExternalAccessible := 'False'; ExternalVisible := 'False'; ExternalWritable := 'False'} : "LSql_typeErrorToken";
   END_VAR

   VAR_IN_OUT 
      tdsTelegramArray : Array[*] of Byte;   // array of bytes received by TDS
      columns : Array[*] of "LSql_typeColumn";
   END_VAR

   VAR 
      statDone { ExternalAccessible := 'False'; ExternalVisible := 'False'; ExternalWritable := 'False'} : Bool;   // static value for output 'done'
      statError { ExternalAccessible := 'False'; ExternalVisible := 'False'; ExternalWritable := 'False'} : Bool;   // static value or output 'error'
      statBusy { ExternalAccessible := 'False'; ExternalVisible := 'False'; ExternalWritable := 'False'} : Bool;   // static value for output 'busy'
      statRowsAvailable { ExternalAccessible := 'False'; ExternalVisible := 'False'; ExternalWritable := 'False'} : Bool;   // static value for output 'metaDataAndRowsAvailable' - Rows available
      statMetaDataAvailable { ExternalAccessible := 'False'; ExternalVisible := 'False'; ExternalWritable := 'False'} : Bool;   // static value for output 'metaDataAndRowsAvailable' - ColumnMetaData available
   END_VAR

   VAR_TEMP 
      tempDeserializePOS : DInt;   // temorary output value of Deserialize function
      tempByteCharArray : Array[0..507] of Byte;   // temporary array of Byte to be transformed to String
      tempTypeLengthOffset : USInt;   // byte address offset for additional length information of data type
      tempColumnSizeFieldSize : USInt;   // size of the area to encode the size of a a value in that column
      tempColumnSize : UDInt;   // size of a value in that column
      tempMoveBlkVariantRetVal : Int;   // return value of MOVE_BLK_VARIANT
      tempTokenEndStatus : UInt;   // temporary value for status to end token
      tempTokenType : Byte;   // temporary value for calculating token type
      tempTableNameParts : USInt;   // number of table name parts in ColumnMeataData
      tempTableNameLength : UInt;   // length of table name parts read from ColumnMetaData
      tempTableNameTotalLength : UInt;   // total length of table name parts in ColumnMetaData
      tempTableNamePartCounter : USInt;   // temporary counter for iteration through able name parts in ColumnMetaData
      tempTableNameByteCounter : DInt;   // comulative counter for Byte address of table name parts in TDS telegram array
      tempRowDataTextptrLen : USInt;   // length of additional field 'Textptr' in Row token
      tempRowDataTextTotalLength : UDInt;   // total length of additional fields 'Text' in Row data
      tempByteAddressCounter : DInt;   // incremental byte address counter
      tempTokenLength : UInt;   // temporary total token length
      tempColumnLength : UDInt;   // column size of real data
      tempColumnLoopCounter : UInt;   // iterative loop counter for the columns
   END_VAR

   VAR CONSTANT 
      BYTE_EMPTY : Byte := 16#0;   // empty Byte
      TDS_TOKEN_TYPEFIELDLENGTH : USInt := 1;   // length of the Token Tpye field
      TDS_TOKEN_LENGTHFIELDLENGTH : USInt := 2;   // length of the field for Token length
      TDS_TOKENROW_TOKENTYPE : Byte := 16#D1;   // Token Type of TDS Row Token
      TDS_COLUMNTYPE_TEXT : UInt := 35;   // identifier of SQL column tpye 'TEXT'
      TDS_COLUMNTYPE_NTEXT : UInt := 99;   // identifier of SQL column type 'NTEXT'
      TDS_COLUMNTYPE_VARIANT : UInt := 98;   // identifier of SQL column type 'VARIANT'
      TDS_COLUMNTYPE_VARIANT_MAXLENGTH : UInt := 8009;   // 'MaxLength for an SSVARIANTTYPE is 8009 (8000 for strings).'
      TDS_TOKENROW_DATATEXTTIMESTAMP_LENGTH : USInt := 8;   // length of field 'Data Text timesatmp'
      TDS_COLUMNMETADATA_TOKENTYPE : Byte := 16#81;   // Token Type of TDS ColumnMetaData Token
      TDS_COLUMNMETADATA_STARTPOS : USInt := 3;   // start Byte of ColumneMetaData
      TDS_COLUMNMETADATA_COLUMNCOUNTPOS : USInt := 1;   // start Byte of CoulmnCount
      TDS_COLUMNMETADATA_TOKENTYPEPOS : USInt := 8;   // start Byte of TokenType
      TDS_COLUMNMETADATA_USERTYPEPOSOFFSET : USInt := 3;   // position offset for user type
      TDS_COLUMNMETADATA_COLUMNTYPEPOSOFFSET : USInt := 6;   // position offset for column type
      TDS_COLUMNMETADATA_COLUMNNAMEPOSOFFSET : USInt := 7;   // position offset for column name
      TDS_COLUMNMETADATA_COLUMNFLAGSPOSOFFSET : USInt := 4;   // position offset for column flags
      TDS_COLUMNMETADATA_COLUMNNAMEPOS : USInt := 8;   // position offset for column name
      TDS_COLUMNMETADATA_FLAGS_NULLABLE : Byte := B#2#0000_0001;   // pattern mask for flag 'nullable'
      TDS_COLUMNMETADATA_FLAGS_CASESENSITIVE : Byte := B#2#0000_0010;   // pattern mask for flag 'case sensitive'
      TDS_COLUMNMETADATA_FLAGS_UPDATEABLE_MASK1100 : Byte := B#2#0000_1100;   // pattern mask for flag 'updateable'
      TDS_COLUMNMETADATA_FLAGS_UPDATEABLE_MASK1000 : Byte := B#2#0000_1000;   // pattern mask for flag 'updateable'
      TDS_COLUMNMETADATA_FLAGS_UPDATEABLE_MASK0100 : Byte := B#2#0000_0100;   // pattern mask for flag 'updateable'
      TDS_COLUMNMETADATA_FLAGS_UPDATEABLE_READONLY : USInt := 0;   // flag value for column is read-only
      TDS_COLUMNMETADATA_FLAGS_UPDATEABLE_READWRITE : USInt := 1;   // flag value for column is read+write
      TDS_COLUMNMETADATA_FLAGS_UPDATEABLE_UNKNOWN : USInt := 2;   // flag value for column access right unknown
      TDS_COLUMNMETADATA_FLAGS_IDENTITY : Byte := B#2#0001_0000;   // pattern mask for flag 'identity'
      TDS_COLUMNMETADATA_FLAGS_COMPUTED : Byte := B#2#0010_0000;   // pattern mask for flag 'computed'
      TDS_COLUMNMETADATA_COLLATELENGTH : USInt := 5;   // byte length of additional collation values (codepage + flags + charset)
      TDS_HEADER_TYPEPOS : USInt := 0;   // byte position in TDS header for 'Type'
      TDS_HEADER_STATUSPOS : USInt := 1;   // byte position in TDS header for 'Status'
      TDS_HEADER_STATUSGOOD : Byte := 16#01;   // value for TDS header status 'Good'
      TDS_HEADER_LENGTHPOS : USInt := 2;   // byte position in TDS header for 'Length'
      TDS_HEADER_SPIDPOS : USInt := 4;   // byte position in TDS header for 'SPID'
      TDS_HEADER_PACKETIDPOS : USInt := 6;   // byte position in TDS header for 'PacketID'
      TDS_HEADER_WINDOWPOS : USInt := 7;   // byte position in TDS header for 'Window'
      TDS_HEADER_LENGTH : USInt := 8;   // length of TDS header
      TDS_COLUMN_SIZEFIELDSIZE_0 : USInt := 0;   // size information is in field of size 0 byte
      TDS_COLUMN_SIZEFIELDSIZE_1 : USInt := 1;   // size information is in field of size 1 byte
      TDS_COLUMN_SIZEFIELDSIZE_2 : USInt := 2;   // size information is in field of size 2 byte
      TDS_COLUMN_SIZEFIELDSIZE_4 : USInt := 4;   // size information is in field of size 4 byte
      TDS_COLUMN_SIZEFIELDSIZE_8 : USInt := 8;   // size information is in field of size 8 byte
      TDS_COLUMN_SIZE_1 : USInt := 1;   // column value size of 1 byte
      TDS_COLUMN_SIZE_2 : USInt := 2;   // column value size of 2 byte
      TDS_COLUMN_SIZE_4 : USInt := 4;   // column value size of 4 byte
      TDS_COLUMN_SIZE_4_MAXVALUE : UDInt := 16#7FFFFFFE;   // column value size of 4 byte
      TDS_COLUMN_SIZE_8 : USInt := 8;   // column value size of 8 byte
      TDS_TOKENDONE_TOKENTYPE : Byte := 16#FD;   // TokenType of TDS Done Token
      TDS_TOKENDONE_STATUSDONEFINAL : UInt := 16#00;   // 'This DONE is the final DONE in the request.'
      TDS_TOKENDONE_STATUSDONEMORE : UInt := 16#01;   // 'This DONE message is not the final DONE message in the response. Subsequent data streams to follow.'
      TDS_TOKENDONE_STATUSDONEERROR : UInt := 16#02;   // 'An error occurred on the current SQL statement. A preceding ERROR token SHOULD be sent when this bit is set.'
      TDS_TOKENDONE_STATUSDONEINXACT : UInt := 16#04;   // 'A transaction is in progress.'
      TDS_TOKENDONE_STATUSDONECOUNT : UInt := 16#10;   // 'The DoneRowCount value is valid. This is used to distinguish between a valid value of 0 for DoneRowCount or just an initialized variable.'
      TDS_TOKENDONE_STATUSDONEATTN : UInt := 16#20;   // 'The DONE message is a server acknowledgement of a client ATTENTION message.'
      TDS_TOKENDONE_STATUSDONESRVERROR : UInt := 16#100;   // Used in place of DONE_ERROR when an error occurred on the current SQL statement, which is severe enough to require the result set, if any, to be discarded.
      TDS_TOKENDONE_STATUSDONE_ROWCOUNTPOS : USInt := 5;   // byte position of RowCount in Done Token
      TDS_TOKENDONE_LENGTH : USInt := 13;   // length of a Done Token
      TDS_TOKENERROR_TOKENTYPE : Byte := 16#AA;   // tokenType of TDS Error Token
      TDS_TOKENERROR_TOKENLENGTHPOS : USInt := 1;   // byte position in Error Token for 'TokenLength'
      TDS_TOKENERROR_SQLERRORNUMBERPOS : USInt := 3;   // byte position in Error Token for 'SQLErrorNumber'
      TDS_TOKENERROR_STATEPOS : USInt := 7;   // byte position in Error Token for 'State'
      TDS_TOKENERROR_CLASSPOS : USInt := 8;   // byte position in Error Token for 'Class'
      TDS_TOKENERROR_ERRORMESSAGELENGTHPOS : USInt := 9;   // byte position in Error Token for 'ErrorMessageLength'
      TDS_TOKENERROR_ERRORMESSAGELENGTHLENGTH : USInt := 2;   // byte length in Error Token for 'ErrorMessageLength'
      TDS_TOKENERROR_SERVERNAMELENGTHLENGTH : USInt := 1;   // byte length in Error Token for 'ServerNameLength'
      TDS_TOKENERROR_PROCNAMELENGTHLENGTH : USInt := 1;   // byte length in Error Token for 'ProcNameLength'
      TDS_TOKENERROR_LINENUMBERLENGTH : USInt := 4;   // byte length in Error Token for 'LineNumber' (documenation says 2 or 8 byte)
      TDS_TOKENDONEINPROC_TOKENTYPE : Byte := 16#FF;   // token type of a TDS DoneInProc Token
      TDS_TOKENDONEINPROC_LENGTH : USInt := 13;   // length of a DoneInProc Token
      TDS_TOKENDONEINPROC_ROWCOUNTPOS : USInt := 5;   // position of value for row count in DoneInProc Token
      TDS_TOKENRETURNSTATUS_TOKENTYPE : Byte := 16#79;   // token type of ReturnStatus Token
      TDS_TOKENRETURNSTATUS_LENGTH : USInt := 5;   // length of ReturnStatus Token
      TDS_TOKENDONEPROC_TOKENTYPE : Byte := 16#FE;   // token type of DoneProc Token
      TDS_TOKENDONEPROC_LENGTH : USInt := 13;   // length of DoneProc Token
      TDS_TOKENENVCHANGE_TOKENTYPE : Byte := 16#E3;   // token type of EnvChange Token
      TDS_TOKENINFO_TOKENTYPE : Byte := 16#AB;   // token type of Info Token
      TDS_TOKENORDER_TOKENTYPE : Byte := 16#A9;   // length of Order Token
      ERR_NOERROR : Word := 16#0000;   // No Error.
      ERR_UNKNOWNTOKEN : Word := 16#8601;   // Error: Unknown Token Type.
      ERR_HEADER_INCORRECTLENGTH : Word := 16#8602;   // Error: Incorrect length in response header.
      ERR_COLUMNS_SIZENOTDEFINED : Word := 16#8603;   // Error: At least one column size is not defined.
      ERR_COLUMNS_TYPENOTDEFINED : Word := 16#8604;   // Error: At least one column type is not defined or unknown.
      ERR_COLUMNS_OVERFLOW : Word := 16#8605;   // Error: Column overflow.
      ERR_TOKENDONE_UNKNOWNSTATUS : Word := 16#8606;   // Error: 'Done' Token has unknown status.
      ERR_TOKENDONE_WRONGTOKENTYPE : Word := 16#8607;   // Error: 'Done' token has wrong Token Type. (outdated)
      ERR_HEADER_WRONGSTATUS : Word := 16#8608;   // Error: Wrong Status in TDS header.
      ERR_TOKENERROR : Word := 16#8609;   // Error: 'Error' Token detected.
      ERR_TOKENROW_NOMETADATA : Word := 16#8610;   // Error: No ColumnMetaData decoded for decoding token row.
      ERR_LENGTHINCORRECT : Word := 16#8611;   // Error: Length of analyzed bytes not matching total TDS telegram length.
      ERR_TYPESIZEINCORRECT : Word := 16#8612;   // Error: A Type Size is incorrect or exceeding the internal array boundaries.
   END_VAR


BEGIN
	REGION BLOCK INFO HEADER
	  //=============================================================================
	  // Siemens AG (c)Copyright (2022)
	  //-----------------------------------------------------------------------------
	  // Library:       SQL
	  // Target:        S7-1500 V2.9 / S7-1200 V4.5
	  // Engineering:   TIA Portal V17
	  // Restrictions:  no
	  // Requirements:  S7-1500 CPU / S7-1200 CPU
	  // Functionality: split SELECT data array from SQL into TDS header, Tokens (especially ColumnMetaData and Error Token) and row payload data
	  //-----------------------------------------------------------------------------
	  // Change log table:
	  // Version    Date         Expert in charge           Changes applied
	  // 01.00.00   31.01.2022   Siemens SUP Applications   initially added to project
	  // 01.00.01   05.07.2022   Siemens SUP Applications   bugfixes:
	  //                                                    - #tempColumnMetaDataByteCounter of type 'USInt' was too short (0-255) --> changed to Datatype 'UInt'
	  //                                                    - #tempColumnSize was not set for columnType 'REAL'
	  //                                                    - #ERR_COLUMNS_OVERFLOW was not checked correctly (#columnCount compared to "NUMBER_OF_COLUMNS")
	  // 01.01.00   06.07.2022   Siemens SUP Applications   added analyzing of Error Token (e.g. after an INSERT command)
	  // 01.02.00   29.09.2022   Siemens SUP Applications   - improved program logic for flexible analyzing of any combination of Tokens
	  //                                                    - added additional TokenTypes: DoneInProc, DoneProc, ResultStatus, Info, EnvChange, Order
	  //                                                    - activated IEC check and adapted formatting
	  //                                                    - including LGF functions for value transformations from Bytes
	  //                                                    - deleted section for clearing unused columns because the number of valid columns is given explicitly
	  // 01.03.00   06.10.2022   Siemens SUP Applications   using FC 'Lsql_BytesToString' for transforming character-based bytes to String                                            
	  //=============================================================================
	END_REGION
	
	//check execute flag
	IF (#execute AND NOT #statDone AND NOT #statError) THEN
	  
	  REGION Execution
	    
	    REGION reset ouput values
	      #statError := FALSE;
	      #statBusy := TRUE;
	      #statDone := FALSE;
	      #statRowsAvailable := FALSE;
	      #statMetaDataAvailable := FALSE;
	      #status := #ERR_NOERROR;
	      #rowCount := 0;
	      #rowDataStart := 0;
	      #rowDataLength := 0;
	      #columnCount := 0;
	      
	      #errorToken.Class := 0;
	      #errorToken.ErrorMessage := '';
	      #errorToken.ErrorMessageLength := 0;
	      #errorToken.LineNumber := 0;
	      #errorToken.ProcName := '';
	      #errorToken.ProcNameLength := 0;
	      #errorToken.ServerName := '';
	      #errorToken.ServerNameLength := 0;
	      #errorToken.SQLErrorNumber := 0;
	      #errorToken.State := 0;
	      #errorToken.TokenLength := 0;
	    END_REGION reset ouput values
	    
	    REGION Header
	      //deserialize 8 byte header information onto tdsHeader
	      #tdsHeader.type := #tdsTelegramArray[#TDS_HEADER_TYPEPOS];
	      #tdsHeader.status := #tdsTelegramArray[#TDS_HEADER_STATUSPOS];
	      #tdsHeader.length := WORD_TO_UINT("LGF_MergeBytesToWord"(byte0 := #tdsTelegramArray[#TDS_HEADER_LENGTHPOS + 1], byte1 := #tdsTelegramArray[#TDS_HEADER_LENGTHPOS]));
	      #tdsHeader.spId.%B1 := #tdsTelegramArray[#TDS_HEADER_SPIDPOS];
	      #tdsHeader.spId.%B0 := #tdsTelegramArray[#TDS_HEADER_SPIDPOS + 1];
	      #tdsHeader.packetID := #tdsTelegramArray[#TDS_HEADER_PACKETIDPOS];
	      #tdsHeader.window := #tdsTelegramArray[#TDS_HEADER_WINDOWPOS];
	      
	      //increment byte position
	      #tempByteAddressCounter := #TDS_HEADER_LENGTH;
	      
	      //check header values
	      IF #tdsHeader.length <= 0 THEN
	        //length value in header is incorrect
	        #status := #ERR_HEADER_INCORRECTLENGTH;
	        #statError := TRUE;
	        #statBusy := FALSE;
	        GOTO END;
	      ELSIF NOT #tdsHeader.status = #TDS_HEADER_STATUSGOOD THEN
	        //status value in header is incorrect
	        #status := #ERR_HEADER_WRONGSTATUS;
	        #statError := TRUE;
	        #statBusy := FALSE;
	        GOTO END;
	      END_IF;
	      
	    END_REGION Header
	    
	    REGION Tokens
	      
	      //loop through all availabe bytes
	      WHILE #tempByteAddressCounter < #tdsHeader.length DO
	        
	        //get Token Type of current token
	        #tempTokenType := #tdsTelegramArray[#tempByteAddressCounter];
	        
	        //case selection depending on Token Type
	        CASE #tempTokenType OF
	            
	          #TDS_COLUMNMETADATA_TOKENTYPE:
	            REGION Token - ColumnMetaData
	              
	              REGION column count
	                //column count is on 1st and 2nd byte
	                #columnCount := WORD_TO_UINT("LGF_MergeBytesToWord"(byte0 := #tdsTelegramArray[#tempByteAddressCounter + #TDS_COLUMNMETADATA_COLUMNCOUNTPOS], byte1 := #tdsTelegramArray[#tempByteAddressCounter + #TDS_COLUMNMETADATA_COLUMNCOUNTPOS + 1]));
	                
	                //check size of column collection to be big enough for all received columns
	                IF #columnCount > ("LSQL_NUMBER_OF_COLUMNS_MAX" + 1) THEN
	                  #status := #ERR_COLUMNS_OVERFLOW;
	                  #statError := TRUE;
	                  GOTO END;
	                END_IF;
	              END_REGION column count
	              
	              REGION columns
	                //jump to start of column data
	                #tempByteAddressCounter += #TDS_COLUMNMETADATA_STARTPOS;
	                
	                //iteration over all column items in tdscolumnMetaData.columns
	                FOR #tempColumnLoopCounter := 0 TO "LSQL_NUMBER_OF_COLUMNS_MAX" BY 1
	                DO
	                  //check if number of columns from SELECT is higher than current iteration index
	                  IF (#tempColumnLoopCounter < #columnCount) THEN
	                    
	                    REGION user type
	                      //get user type of current column
	                      #columns[#tempColumnLoopCounter].userType := BYTE_TO_UDINT(#tdsTelegramArray[#tempByteAddressCounter + #TDS_COLUMNMETADATA_USERTYPEPOSOFFSET]);
	                    END_REGION user type
	                    
	                    REGION flags
	                      //get column properties flags by bit masquerading as additional information about current column
	                      
	                      //property 'nullable'
	                      #columns[#tempColumnLoopCounter].flags.nullable := ((#tdsTelegramArray[#tempByteAddressCounter + #TDS_COLUMNMETADATA_COLUMNFLAGSPOSOFFSET] AND #TDS_COLUMNMETADATA_FLAGS_NULLABLE) > 0);
	                      //property 'caseSensitive'
	                      #columns[#tempColumnLoopCounter].flags.caseSensitive := ((#tdsTelegramArray[#tempByteAddressCounter + #TDS_COLUMNMETADATA_COLUMNFLAGSPOSOFFSET] AND #TDS_COLUMNMETADATA_FLAGS_CASESENSITIVE) > 0);
	                      
	                      //property 'updateable'
	                      IF ((#tdsTelegramArray[#tempByteAddressCounter + #TDS_COLUMNMETADATA_COLUMNFLAGSPOSOFFSET] AND #TDS_COLUMNMETADATA_FLAGS_UPDATEABLE_MASK1100) > 0) THEN
	                        #columns[#tempColumnLoopCounter].flags.updateable := #TDS_COLUMNMETADATA_FLAGS_UPDATEABLE_UNKNOWN;
	                      ELSIF ((#tdsTelegramArray[#tempByteAddressCounter + #TDS_COLUMNMETADATA_COLUMNFLAGSPOSOFFSET] AND #TDS_COLUMNMETADATA_FLAGS_UPDATEABLE_MASK0100) > 0) THEN
	                        #columns[#tempColumnLoopCounter].flags.updateable := #TDS_COLUMNMETADATA_FLAGS_UPDATEABLE_READWRITE;
	                      ELSIF ((#tdsTelegramArray[#tempByteAddressCounter + #TDS_COLUMNMETADATA_COLUMNFLAGSPOSOFFSET] AND #TDS_COLUMNMETADATA_FLAGS_UPDATEABLE_MASK1000) > 0) THEN
	                        #columns[#tempColumnLoopCounter].flags.updateable := #TDS_COLUMNMETADATA_FLAGS_UPDATEABLE_UNKNOWN;
	                      ELSE
	                        #columns[#tempColumnLoopCounter].flags.updateable := #TDS_COLUMNMETADATA_FLAGS_UPDATEABLE_READONLY;
	                      END_IF;
	                      
	                      //property 'identity'
	                      #columns[#tempColumnLoopCounter].flags.identity := ((#tdsTelegramArray[#tempByteAddressCounter + #TDS_COLUMNMETADATA_COLUMNFLAGSPOSOFFSET] AND #TDS_COLUMNMETADATA_FLAGS_IDENTITY) > 0);
	                      //property 'computed'
	                      #columns[#tempColumnLoopCounter].flags.computed := ((#tdsTelegramArray[#tempByteAddressCounter + #TDS_COLUMNMETADATA_COLUMNFLAGSPOSOFFSET] AND #TDS_COLUMNMETADATA_FLAGS_COMPUTED) > 0);
	                    END_REGION flags
	                    
	                    REGION column type
	                      //get column type as important information about data type and encoding sizes
	                      
	                      #columns[#tempColumnLoopCounter].columnType := BYTE_TO_UINT(IN := #tdsTelegramArray[#tempByteAddressCounter + #TDS_COLUMNMETADATA_COLUMNTYPEPOSOFFSET]);
	                    END_REGION column type
	                    
	                    REGION type length
	                      //read or set type lengths depending on columnType:
	                      //e.g. columnType '56' means 'INT4': value field size is not given in telegram data (#tempColumnSizeFieldSize := 0) because value always has a size of 4 byte (#tempColumnSize := 4)
	                      //e.g. columnType '167' means 'VARCHAR': value field size is given in 2 additional byte (#tempColumnSizeFieldSize := 2) in which the size (#tempColumnSize) of the string will be given
	                      //
	                      //table source:
	                      //https://www.freetds.org/tds.html#types
	                      
	                      #tempColumnSize := 0;
	                      
	                      CASE #columns[#tempColumnLoopCounter].columnType OF
	                        31://VOID
	                          #tempColumnSizeFieldSize := #TDS_COLUMN_SIZEFIELDSIZE_0;
	                          #tempTypeLengthOffset := #tempColumnSizeFieldSize;
	                        34://IMAGE
	                          #tempColumnSizeFieldSize := #TDS_COLUMN_SIZEFIELDSIZE_4;
	                          #tempTypeLengthOffset := #tempColumnSizeFieldSize;
	                        #TDS_COLUMNTYPE_TEXT://35 - TEXT
	                          #tempColumnSizeFieldSize := #TDS_COLUMN_SIZEFIELDSIZE_4;
	                          
	                          REGION Table Names
	                            #tempTableNameByteCounter := #tempByteAddressCounter + USINT_TO_DINT(IN := #TDS_COLUMNMETADATA_COLUMNTYPEPOSOFFSET) + 1 + USINT_TO_DINT(IN := #tempColumnSizeFieldSize) + #TDS_COLUMNMETADATA_COLLATELENGTH;
	                            
